# B&R Automation Studio project PickAndPlace
Automation Studio 6.3.1.32; Default project; technology packages: mappCockpit 6.3.1, mappMotion 6.4.1, mappView 6.3.1, mappVision 6.0.0, OpcUaCs 6.3.1

## Configuration APC3100

CPU 5APC3100.KBU3-000, AutomationRuntime 6.5.1, Build 11.3.0, Safety 0.0

### Task classes (Cpu.sw)
```
Cyclic#1 (cycle 2000 us, tolerance 0 us):
  Camera <- Tasks.Camera.prg
  BufferInit <- Tasks.BufferInit.prg
  Mechanics <- Tasks.Mechanics.prg
DataObjects: McAcpSys, assl1, Acp10sys, Arnc0sys
NcDataObjects: McDriveLog, gS_AxRepoi, gS_AxR1QCa, gS_AxR1QCi, gS_AxRepoa
Binaries: udbdef, arsvcreg, McMechSys, McAcpSim, McAcpDrv, TCData, mvLoader, McProfGen, mvConfig, OpcUaSrv, ViUnits, mCoWebSc, ashwac, Hierarchy, arconfig, ashwd, asfw, sysconf, iomap, Role, User, Settings, MechSys2, MechSys1, AxGrp1, Feat2, Axis2, Axis1, TrkPath, Feat1, AxGrp2, Ws2, Ws1, Conveyer, Config, Config_1, Config_2, TraceConfi, UaCsConfig, BRRole, Conveyor, TrkFrmSel1, TrkFrmSel2, viComp, Settings_1, viApp, viApp_1, FWRules, Config_3, ArFlatPrv, ArCoal, Config_8, vcpk, vcwxprt, vcpfar10, vcshared, vcfile, vcpfmtcx, arial, vcgclass, vcalarm, vcdsint, vcpfapc, arialbd, vcdsloc, vcmgr, vcbclass, StdVi102, StdVi101, StdVi103, StdVis02, StdVis03, StdVis01, vcnet, vctcal, vcpdihd, vcptusb, acp10cfg, Arnc0map, arnc0cfg, Acp10map, TCPmap, vcfntttf, vccbmp, SimVis01, vcrt, vcpdvnc, SimVis02, vcpdsw, vcpkat, vcctext, SimVis03, vccshape, vccbtn, vccovl, AdvVis03, AdvVis02, AdvVis01, vccstr, vccurl, vccbar, vcchtml, vccnum, vcxml, vccalarm, vcclbox, vccedit, Config_7, Config_6, Config_4, Config_5, TrkPath1
Libraries: Runtime, Operator, AsIecCon, astime, sys_lib, FileIO, AsMem, brsystem, AsBrStr, AsIOTime, standard, AsArSdm, AsBrWStr, AsZip, AsIO, AsHttp, AsIODiag, AsBrMath, MpBase, CoTrace, McBase, McAxGroup, McAcpAx, McAxis, McPathGen, McTrkPath, MpAxis, McProgInt, MpPick, McPureVAx, MpRobotics, MpTool, ViBase, AsARCfg, powerlnk, AsEPL, AsTCP, ArSsl, DataObj, UaCoal, AsArProf, UaCoalPrv, UaCore, ashw, vcresman
```

### Hardware
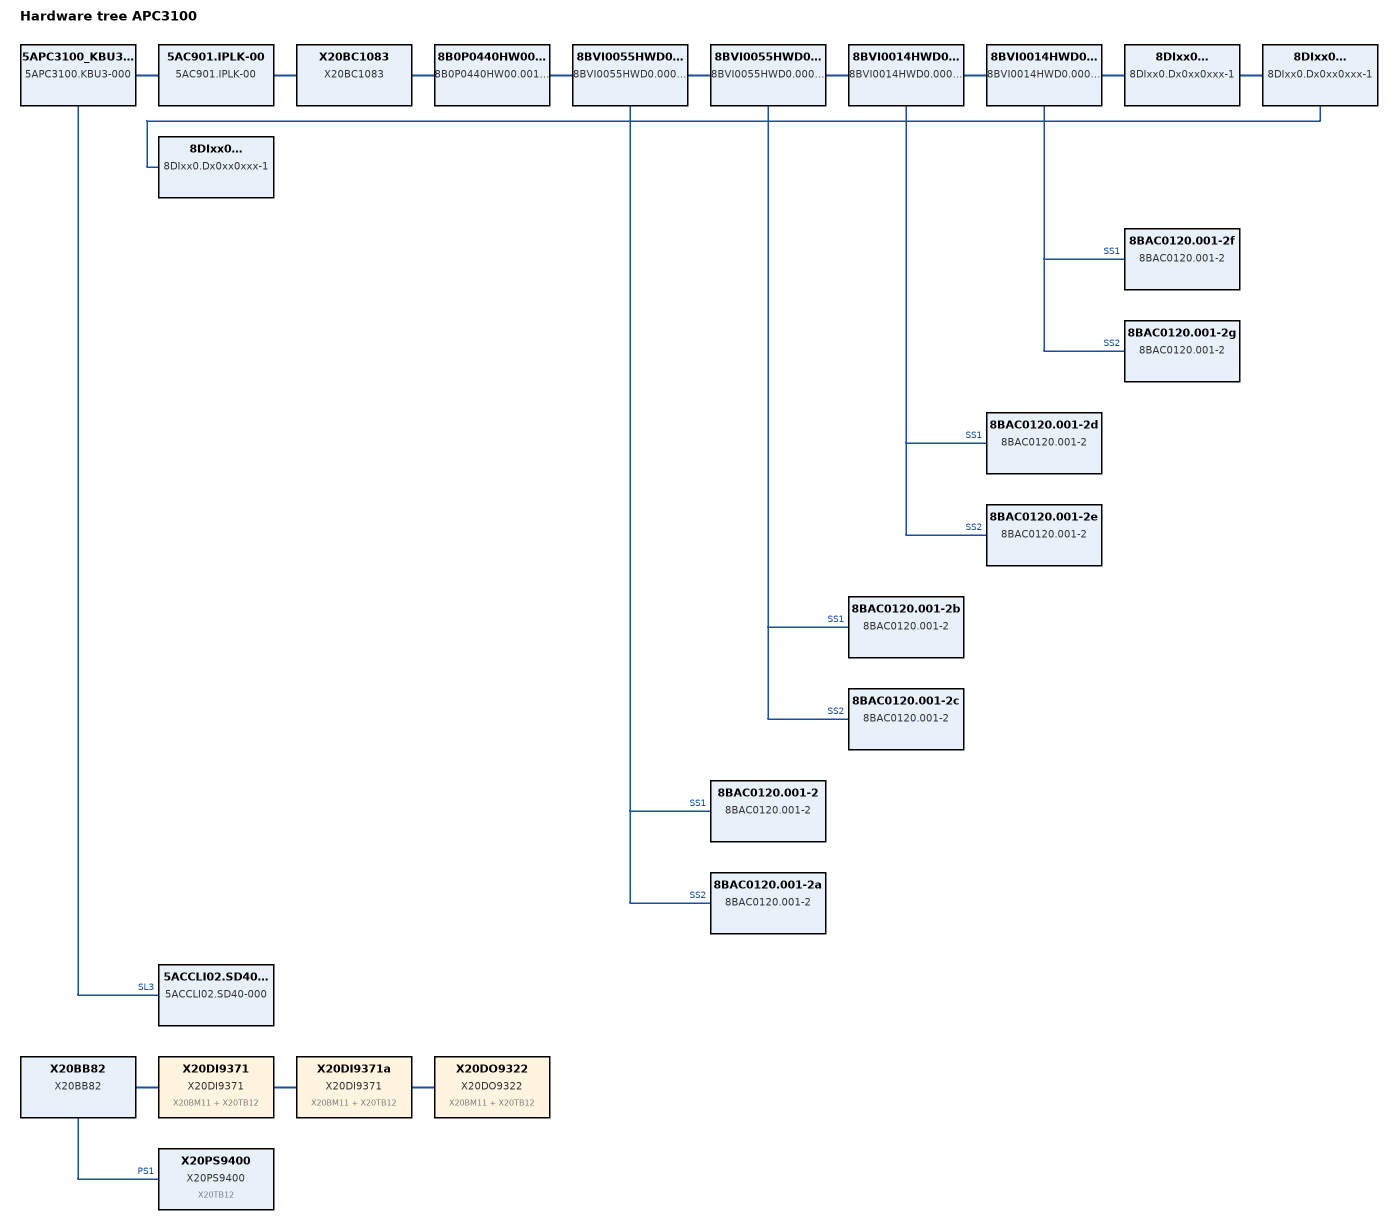
```
5AC901.IPLK-00 : 5AC901.IPLK-00 v2.1.0.0  [SL -> 5APC3100_KBU3_000.SL2]
  Connector IF1:
    MtuSize = 1500
    Channel1
    ChannelID1 = McAcpBroadcast
    ChannelType1 = OCTET[96]
    InternetAddress = 192.168.200.240
    SubnetMask = 255.255.255.0
    ActivateANSL = 1
    ActivateIpForwarding = 1
5ACCLI02.SD40-000 : 5ACCLI02.SD40-000 v2.1.0.0  [SL -> 5APC3100_KBU3_000.SL3]
  Supervision = off
5APC3100_KBU3_000 : 5APC3100.KBU3-000 v2.3.1.0
  Connector IF3:
    AssignedOperatingSystem = ARemb
    ActivateDevice = 1
    HostName = apc3100motorlabsbg
  Connector IF4:
    AssignedOperatingSystem = ARemb
    ActivateDevice = 1
    HostName = apc3100motorlabsbg
    Mode = Manual
    InternetAddress = 192.168.20.250
    SubnetMask = 255.255.255.0
    Vnc1
    VncTitle1 = VNC
    ActivateSnmp = 2
    ActivateIpForwarding = 1
  Connector IF5:
    AssignedOperatingSystem = ARemb
  Connector IF6:
    AssignedOperatingSystem = ARemb
  Connector IF7:
    AssignedOperatingSystem = ARemb
  Connector IF8:
    AssignedOperatingSystem = ARemb
  ConfigurationID = PickAndPlace_Real_APC910
  Simulation = 1
  RemMemDevice = PCI.2.IPLK.SRAM
  RemMemSize = 64000
  PermanentPvSize = 32000
  RemanentGlobalPvSize = 16000
  TimerDeviceType = EPLX2X
  TimerDevice = 5AC901.IPLK-00.IF1
  TaskClassIdleTime = 2000
  Cyclic1Duration = 2000
  Cyclic1Tolerance = 0
  Cyclic1Stack = 655360
  Cyclic1Output = 1
  Cyclic2Duration = 4000
  Cyclic2Tolerance = 4000
  Cyclic3Duration = 6000
  Cyclic3Tolerance = 6000
  Cyclic4Duration = 8000
  Cyclic4Tolerance = 8000
  Cyclic5Duration = 100000
  Cyclic5Tolerance = 100000
  FileDevice1
  FileDeviceName1 = RobotMotionPrgDir
  FileDevicePath1 = USER_PATH\..\..\..\..\..\Logical\UserPartitionData\RobotMotionPrgDir  // No simulation: use  USER_PATH\RobotMotionPrgDir   ;        Simulation: use    USER_PATH\..\..\..\..\..\Logical\UserPartitionData\RobotMotionPrgDir    to directly access the current progam state
  FileDevice2
  FileDeviceName2 = AutoGeneratedScene
  FileDevicePath2 = USER_PATH
  EthernetHostName = apc3100motorlabsbg
  ActivateFtpServer = 1
  FtpUser1
  FtpUsername1 = gmctest
  FtpUserPassword1 = qT0dlrKemp8H+/2V4GRHUzUq1qxdxChn7SWtcolMOPQ=
  FtpUserSalt1 = 1zGWL4Fu
  FTPAccessRight1 = 0
  ActivateWebServer = 1
  ActivateSdm = 1
8B0P0440HW00.001-1 : 8B0P0440HW00.001-1 v2.3.0.3 (NodeNumber=4)  [PLK1 -> X20BC1083.PLK2 [Cable Type=PowerlinkCable, Length=10, Version=1.0.0.3]; PLK2 -> 8BVI0055HWD0.000-1.PLK1 [Cable Type=PowerlinkCable, Length=10, Version=1.0.0.3]]
  DriveConfiguration/Module:
    McAcoposTypeID = AcoposMultiPSMpConfig
    ActivateACOPOSSimulationOnPLC = 0
    SWResetAfterFirmwareUpdate = 0
  DriveConfiguration/Channel[1]/PowerSection:
    AxisReference = gPsm
8BAC0120.001-2 : 8BAC0120.001-2 v2.2.0.0  [SS -> 8BVI0055HWD0.000-1.SS1]  // Delta 1 - Q1
  PlugInType = Encoder
  McAcoposTypeID = AcoposMultiPlugInConfig
8BAC0120.001-2a : 8BAC0120.001-2 v2.2.0.0  [SS -> 8BVI0055HWD0.000-1.SS2]  // Delta 1 - Q3
  PlugInType = Encoder
  McAcoposTypeID = AcoposMultiPlugInConfig
8BAC0120.001-2b : 8BAC0120.001-2 v2.2.0.0  [SS -> 8BVI0055HWD0.000-1a.SS1]  // Delta 1 - Q2
  PlugInType = Encoder
  McAcoposTypeID = AcoposMultiPlugInConfig
8BAC0120.001-2c : 8BAC0120.001-2 v2.2.0.0  [SS -> 8BVI0055HWD0.000-1a.SS2]  // Delta 1 - Qc
  PlugInType = Encoder
  McAcoposTypeID = AcoposMultiPlugInConfig
8BAC0120.001-2d : 8BAC0120.001-2 v2.2.0.0  [SS -> 8BVI0014HWD0.000-1.SS1]  // Delta 2 - Qc
  PlugInType = Encoder
  McAcoposTypeID = AcoposMultiPlugInConfig
8BAC0120.001-2e : 8BAC0120.001-2 v2.2.0.0  [SS -> 8BVI0014HWD0.000-1.SS2]  // Conveyer 1
  PlugInType = Encoder
  McAcoposTypeID = AcoposMultiPlugInConfig
8BAC0120.001-2f : 8BAC0120.001-2 v2.2.0.0  [SS -> 8BVI0014HWD0.000-1a.SS1]  // Conveyer 2
  PlugInType = Encoder
  McAcoposTypeID = AcoposMultiPlugInConfig
8BAC0120.001-2g : 8BAC0120.001-2 v2.2.0.0  [SS -> 8BVI0014HWD0.000-1a.SS2]  // Repository
  PlugInType = Encoder
  McAcoposTypeID = AcoposMultiPlugInConfig
8BVI0014HWD0.000-1 : 8BVI0014HWD0.000-1 v2.3.0.2 (NodeNumber=7)  [PLK1 -> 8BVI0055HWD0.000-1a.PLK2 [Cable Type=PowerlinkCable, Length=10, Version=1.0.0.3]; PLK2 -> 8BVI0014HWD0.000-1a.PLK1 [Cable Type=PowerlinkCable, Length=10, Version=1.0.0.3]]
  DriveConfiguration/Module:
    PowerSupply = DCBusVoltage
  DriveConfiguration/Module/PowerSupply:
    BusVoltage = 550
  DriveConfiguration/Channel[1]/RealAxis:
    AxisReference = delta2Qc
  DriveConfiguration/Channel[1]/RealAxis/MechanicalElements/Gearbox:
    Input = 10
  DriveConfiguration/Channel[1]/RealAxis/MechanicalElements/RotaryToLinearTransformation:
    ReferenceDistance = 3
  DriveConfiguration/Channel[1]/RealAxis/Controller/Mode/Position:
    ProportionalGain = 340
  DriveConfiguration/Channel[1]/RealAxis/Controller/Mode/Speed:
    ProportionalGain = 1.35
  DriveConfiguration/Channel[1]/RealAxis/Homing:
    Mode = Absolute
  DriveConfiguration/Channel[1]/RealAxis/Homing/Mode:
    Position = 14929.177
  DriveConfiguration/Channel[1]/RealAxis/Homing:
    RestorePositionVariable = 
  DriveConfiguration/Channel[1]/RealAxis/MovementErrorLimits:
    PositionError = 1.0
  DriveConfiguration/Channel[2]/RealAxis:
    AxisReference = conveyer1Ax
  DriveConfiguration/Channel[2]/RealAxis/MechanicalElements/Gearbox:
    Output = 10
  DriveConfiguration/Channel[2]/RealAxis/MechanicalElements/RotaryToLinearTransformation:
    ReferenceDistance = 3
  DriveConfiguration/Channel[2]/RealAxis/Controller/Mode/Position:
    ProportionalGain = 460
  DriveConfiguration/Channel[2]/RealAxis/Controller/Mode/Speed:
    ProportionalGain = 0.6
  DriveConfiguration/Channel[2]/RealAxis/Homing/Mode:
    Position = 5
  DriveConfiguration/Channel[2]/RealAxis/Homing:
    RestorePositionVariable = 
  DriveConfiguration/Channel[2]/RealAxis/MovementErrorLimits:
    PositionError = 1.0
  DriveConfiguration/Channel[2]/RealAxis/AxisFeatures:
    FeatureRef[1] = ProfGen
8BVI0014HWD0.000-1a : 8BVI0014HWD0.000-1 v2.3.0.2  [PLK1 -> 8BVI0014HWD0.000-1.PLK2 [Cable Type=PowerlinkCable, Length=10, Version=1.0.0.3]; PLK2 -> 8DIxx0.Dx0xx0xxx-1.PLK1 [Cable Type=PowerlinkCable, Length=10, Version=1.0.0.3]]
  DriveConfiguration/Module:
    PowerSupply = DCBusVoltage
  DriveConfiguration/Module/PowerSupply:
    BusVoltage = 550
  DriveConfiguration/Channel[1]/RealAxis:
    AxisReference = conveyer2Ax
  DriveConfiguration/Channel[1]/RealAxis/MechanicalElements/Gearbox:
    Output = 10
  DriveConfiguration/Channel[1]/RealAxis/MechanicalElements/RotaryToLinearTransformation:
    ReferenceDistance = 3
  DriveConfiguration/Channel[1]/RealAxis/Controller/Mode/Position:
    ProportionalGain = 420
  DriveConfiguration/Channel[1]/RealAxis/Controller/Mode/Speed:
    ProportionalGain = 0.55
  DriveConfiguration/Channel[1]/RealAxis/Homing/Mode:
    Position = 5
  DriveConfiguration/Channel[1]/RealAxis/Homing:
    RestorePositionVariable = 
  DriveConfiguration/Channel[1]/RealAxis/MovementErrorLimits:
    PositionError = 1.0
  DriveConfiguration/Channel[1]/RealAxis/AxisFeatures:
    FeatureRef[1] = ProfGen
  DriveConfiguration/Channel[2]/RealAxis:
    AxisReference = repositoryAx
  DriveConfiguration/Channel[2]/RealAxis/MechanicalElements/RotaryToLinearTransformation:
    ReferenceDistance = 16
  DriveConfiguration/Channel[2]/RealAxis/Controller/Mode/Position:
    ProportionalGain = 500.0
  DriveConfiguration/Channel[2]/RealAxis/Controller/Mode/Speed:
    ProportionalGain = 0.3
  DriveConfiguration/Channel[2]/RealAxis/Homing:
    Mode = Absolute
  DriveConfiguration/Channel[2]/RealAxis/Homing/Mode:
    Position = -58251.071
  DriveConfiguration/Channel[2]/RealAxis/Homing:
    RestorePositionVariable = 
  DriveConfiguration/Channel[2]/RealAxis/MovementErrorLimits:
    PositionError = 1.0
8BVI0055HWD0.000-1 : 8BVI0055HWD0.000-1 v2.3.0.2 (NodeNumber=5)  [PLK1 -> 8B0P0440HW00.001-1.PLK2 [Cable Type=PowerlinkCable, Length=10, Version=1.0.0.3]; PLK2 -> 8BVI0055HWD0.000-1a.PLK1 [Cable Type=PowerlinkCable, Length=10, Version=1.0.0.3]]
  DriveConfiguration/Module:
    McAcoposTypeID = AcoposMultiDConfig
    ActivateACOPOSSimulationOnPLC = 0
    PowerSupply = DCBusVoltage
  DriveConfiguration/Module/PowerSupply:
    BusVoltage = 550
  DriveConfiguration/Channel[1]/RealAxis:
    AxisReference = delta1Q1
    MechanicalElementsIsInvisible = 0
  DriveConfiguration/Channel[1]/RealAxis/MechanicalElements/Gearbox:
    InputIsReadOnly = 0
    Input = 31
    OutputIsReadOnly = 0
    Output = 1
  DriveConfiguration/Channel[1]/RealAxis/MechanicalElements/RotaryToLinearTransformation:
    ReferenceDistanceIsReadOnly = 0
    ReferenceDistance = 1
  DriveConfiguration/Channel[1]/RealAxis/Controller:
    ModeIsReadOnly = 0
    Mode = PositionController
  DriveConfiguration/Channel[1]/RealAxis/Controller/Mode/Position:
    ProportionalGain = 420
    IntegrationTime = 0.0
    PredictionTime = 0.0004
    TotalDelayTime = 0.0004
  DriveConfiguration/Channel[1]/RealAxis/Controller/Mode/Speed:
    ProportionalGainIsReadOnly = 0
    ProportionalGain = 1.65
    IntegrationTimeIsReadOnly = 0
    IntegrationTime = 0.0
    FilterTimeIsReadOnly = 0
    FilterTime = 0.0
  DriveConfiguration/Channel[1]/RealAxis/Controller/Mode/LoopFilters:
    LoopFilterXIsReadOnly = 0
    LoopFilter1 = NotUsed
    LoopFilter2 = NotUsed
    LoopFilter3 = NotUsed
  DriveConfiguration/Channel[1]/RealAxis/Homing:
    ModeIsReadOnly = 0
    Mode = Absolute
  DriveConfiguration/Channel[1]/RealAxis/Homing/Mode:
    Position = 17776.525
  DriveConfiguration/Channel[1]/RealAxis/Homing:
    RestorePositionVariable = 
  DriveConfiguration/Channel[1]/RealAxis/StopReaction:
    QuickstopIsReadOnly = 0
    Quickstop = DecelerationLimit
    DriveErrorIsReadOnly = 0
    DriveError = DecelerationLimit
  DriveConfiguration/Channel[1]/RealAxis/MovementErrorLimits:
    PositionError = 1.0
    VelocityErrorMonitoring = Automatic1
  DriveConfiguration/Channel[1]/RealAxis:
    JerkFilterIsReadOnly = 0
    JerkFilter = NotUsed
    ZeroVibrationFilter = NotUsed
  DriveConfiguration/Channel[1]/RealAxis/DigitalInputs/HomingSwitch:
    SourceIsReadOnly = 0
    Source = NotUsed
    Level = High
  DriveConfiguration/Channel[1]/RealAxis/DigitalInputs/PositiveLimitSwitch:
    SourceIsReadOnly = 0
    Source = NotUsed
    Level = High
  DriveConfiguration/Channel[1]/RealAxis/DigitalInputs/NegativeLimitSwitch:
    SourceIsReadOnly = 0
    Source = NotUsed
    Level = High
  DriveConfiguration/Channel[1]/RealAxis/DigitalInputs/Trigger1:
    Source = X2Trigger1
    Level = High
  DriveConfiguration/Channel[1]/RealAxis/DigitalInputs/Trigger2:
    Source = X2Trigger2
    Level = High
  DriveConfiguration/Channel[1]/RealAxis/DigitalInputs/Quickstop:
    Input = Trigger2
  DriveConfiguration/Channel[1]/RealAxis/Simulation:
    SimulationModeOnPLC = SetValueGeneration
    SimulationModeOnACOPOS = NotUsed
  DriveConfiguration/Channel[1]:
    ExternalEncoderAxis = NotUsed
  DriveConfiguration/Channel[2]/RealAxis:
    AxisReference = delta1Q3
    MechanicalElementsIsInvisible = 0
  DriveConfiguration/Channel[2]/RealAxis/MechanicalElements/Gearbox:
    InputIsReadOnly = 0
    Input = 31
    OutputIsReadOnly = 0
    Output = 1
  DriveConfiguration/Channel[2]/RealAxis/MechanicalElements/RotaryToLinearTransformation:
    ReferenceDistanceIsReadOnly = 0
    ReferenceDistance = 1
  DriveConfiguration/Channel[2]/RealAxis/Controller:
    ModeIsReadOnly = 0
    Mode = PositionController
  DriveConfiguration/Channel[2]/RealAxis/Controller/Mode/Position:
    ProportionalGain = 420
    IntegrationTime = 0.0
    PredictionTime = 0.0004
    TotalDelayTime = 0.0004
  DriveConfiguration/Channel[2]/RealAxis/Controller/Mode/Speed:
    ProportionalGainIsReadOnly = 0
    ProportionalGain = 1.65
    IntegrationTimeIsReadOnly = 0
    IntegrationTime = 0.0
    FilterTimeIsReadOnly = 0
    FilterTime = 0.0
  DriveConfiguration/Channel[2]/RealAxis/Controller/Mode/LoopFilters:
    LoopFilterXIsReadOnly = 0
    LoopFilter1 = NotUsed
    LoopFilter2 = NotUsed
    LoopFilter3 = NotUsed
  DriveConfiguration/Channel[2]/RealAxis/Homing:
    ModeIsReadOnly = 0
    Mode = Absolute
  DriveConfiguration/Channel[2]/RealAxis/Homing/Mode:
    Position = 44644.06
  DriveConfiguration/Channel[2]/RealAxis/Homing:
    RestorePositionVariable = 
  DriveConfiguration/Channel[2]/RealAxis/StopReaction:
    QuickstopIsReadOnly = 0
    Quickstop = DecelerationLimit
    DriveErrorIsReadOnly = 0
    DriveError = DecelerationLimit
  DriveConfiguration/Channel[2]/RealAxis/MovementErrorLimits:
    PositionError = 1.0
    VelocityErrorMonitoring = Automatic1
  DriveConfiguration/Channel[2]/RealAxis:
    JerkFilterIsReadOnly = 0
    JerkFilter = NotUsed
    ZeroVibrationFilter = NotUsed
  DriveConfiguration/Channel[2]/RealAxis/DigitalInputs/HomingSwitch:
    SourceIsReadOnly = 0
    Source = NotUsed
    Level = High
  DriveConfiguration/Channel[2]/RealAxis/DigitalInputs/PositiveLimitSwitch:
    SourceIsReadOnly = 0
    Source = NotUsed
    Level = High
  DriveConfiguration/Channel[2]/RealAxis/DigitalInputs/NegativeLimitSwitch:
    SourceIsReadOnly = 0
    Source = NotUsed
    Level = High
  DriveConfiguration/Channel[2]/RealAxis/DigitalInputs/Trigger1:
    Source = X2Trigger1
    Level = High
  DriveConfiguration/Channel[2]/RealAxis/DigitalInputs/Trigger2:
    Source = X2Trigger2
    Level = High
  DriveConfiguration/Channel[2]/RealAxis/DigitalInputs/Quickstop:
    Input = Trigger2
  DriveConfiguration/Channel[2]/RealAxis/Simulation:
    SimulationModeOnPLC = SetValueGeneration
    SimulationModeOnACOPOS = NotUsed
  DriveConfiguration/Channel[2]:
    ExternalEncoderAxis = NotUsed
8BVI0055HWD0.000-1a : 8BVI0055HWD0.000-1 v2.3.0.2 (NodeNumber=6)  [PLK1 -> 8BVI0055HWD0.000-1.PLK2 [Cable Type=PowerlinkCable, Length=10, Version=1.0.0.3]; PLK2 -> 8BVI0014HWD0.000-1.PLK1 [Cable Type=PowerlinkCable, Length=10, Version=1.0.0.3]]
  DriveConfiguration/Module:
    McAcoposTypeID = AcoposMultiDConfig
    ActivateACOPOSSimulationOnPLC = 0
    PowerSupply = DCBusVoltage
  DriveConfiguration/Module/PowerSupply:
    BusVoltage = 550
  DriveConfiguration/Channel[1]/RealAxis:
    AxisReference = delta1Q2
    MechanicalElementsIsInvisible = 0
  DriveConfiguration/Channel[1]/RealAxis/MechanicalElements/Gearbox:
    InputIsReadOnly = 0
    Input = 31
    OutputIsReadOnly = 0
    Output = 1
  DriveConfiguration/Channel[1]/RealAxis/MechanicalElements/RotaryToLinearTransformation:
    ReferenceDistanceIsReadOnly = 0
    ReferenceDistance = 1
  DriveConfiguration/Channel[1]/RealAxis/Controller:
    ModeIsReadOnly = 0
    Mode = PositionController
  DriveConfiguration/Channel[1]/RealAxis/Controller/Mode/Position:
    ProportionalGain = 420
    IntegrationTime = 0.0
    PredictionTime = 0.0004
    TotalDelayTime = 0.0004
  DriveConfiguration/Channel[1]/RealAxis/Controller/Mode/Speed:
    ProportionalGainIsReadOnly = 0
    ProportionalGain = 1.65
    IntegrationTimeIsReadOnly = 0
    IntegrationTime = 0.0
    FilterTimeIsReadOnly = 0
    FilterTime = 0.0
  DriveConfiguration/Channel[1]/RealAxis/Controller/Mode/LoopFilters:
    LoopFilterXIsReadOnly = 0
    LoopFilter1 = NotUsed
    LoopFilter2 = NotUsed
    LoopFilter3 = NotUsed
  DriveConfiguration/Channel[1]/RealAxis/Homing:
    ModeIsReadOnly = 0
    Mode = Absolute
  DriveConfiguration/Channel[1]/RealAxis/Homing/Mode:
    Position = 26128.766
  DriveConfiguration/Channel[1]/RealAxis/Homing:
    RestorePositionVariable = 
  DriveConfiguration/Channel[1]/RealAxis/StopReaction:
    QuickstopIsReadOnly = 0
    Quickstop = DecelerationLimit
    DriveErrorIsReadOnly = 0
    DriveError = DecelerationLimit
  DriveConfiguration/Channel[1]/RealAxis/MovementErrorLimits:
    PositionError = 1.0
    VelocityErrorMonitoring = Automatic1
  DriveConfiguration/Channel[1]/RealAxis:
    JerkFilterIsReadOnly = 0
    JerkFilter = NotUsed
    ZeroVibrationFilter = NotUsed
  DriveConfiguration/Channel[1]/RealAxis/DigitalInputs/HomingSwitch:
    SourceIsReadOnly = 0
    Source = NotUsed
    Level = High
  DriveConfiguration/Channel[1]/RealAxis/DigitalInputs/PositiveLimitSwitch:
    SourceIsReadOnly = 0
    Source = NotUsed
    Level = High
  DriveConfiguration/Channel[1]/RealAxis/DigitalInputs/NegativeLimitSwitch:
    SourceIsReadOnly = 0
    Source = NotUsed
    Level = High
  DriveConfiguration/Channel[1]/RealAxis/DigitalInputs/Trigger1:
    Source = X2Trigger1
    Level = High
  DriveConfiguration/Channel[1]/RealAxis/DigitalInputs/Trigger2:
    Source = X2Trigger2
    Level = High
  DriveConfiguration/Channel[1]/RealAxis/DigitalInputs/Quickstop:
    Input = Trigger2
  DriveConfiguration/Channel[1]/RealAxis/Simulation:
    SimulationModeOnPLC = SetValueGeneration
    SimulationModeOnACOPOS = NotUsed
  DriveConfiguration/Channel[1]:
    ExternalEncoderAxis = NotUsed
  DriveConfiguration/Channel[2]/RealAxis:
    AxisReference = delta1Qc
    MechanicalElementsIsInvisible = 0
  DriveConfiguration/Channel[2]/RealAxis/MechanicalElements/Gearbox:
    InputIsReadOnly = 0
    Input = 10
    OutputIsReadOnly = 0
    Output = 1
  DriveConfiguration/Channel[2]/RealAxis/MechanicalElements/RotaryToLinearTransformation:
    ReferenceDistanceIsReadOnly = 0
    ReferenceDistance = 1
  DriveConfiguration/Channel[2]/RealAxis/Controller:
    ModeIsReadOnly = 0
    Mode = PositionController
  DriveConfiguration/Channel[2]/RealAxis/Controller/Mode/Position:
    ProportionalGain = 400
    IntegrationTime = 0.0
    PredictionTime = 0.0004
    TotalDelayTime = 0.0004
  DriveConfiguration/Channel[2]/RealAxis/Controller/Mode/Speed:
    ProportionalGainIsReadOnly = 0
    ProportionalGain = 1.2
    IntegrationTimeIsReadOnly = 0
    IntegrationTime = 0.0
    FilterTimeIsReadOnly = 0
    FilterTime = 0.0
  DriveConfiguration/Channel[2]/RealAxis/Controller/Mode/LoopFilters:
    LoopFilterXIsReadOnly = 0
    LoopFilter1 = NotUsed
    LoopFilter2 = NotUsed
    LoopFilter3 = NotUsed
  DriveConfiguration/Channel[2]/RealAxis/Homing:
    ModeIsReadOnly = 0
    Mode = Absolute
  DriveConfiguration/Channel[2]/RealAxis/Homing/Mode:
    Position = 68668.338
  DriveConfiguration/Channel[2]/RealAxis/Homing:
    RestorePositionVariable = 
  DriveConfiguration/Channel[2]/RealAxis/StopReaction:
    QuickstopIsReadOnly = 0
    Quickstop = DecelerationLimit
    DriveErrorIsReadOnly = 0
    DriveError = DecelerationLimit
  DriveConfiguration/Channel[2]/RealAxis/MovementErrorLimits:
    PositionError = 1.0
    VelocityErrorMonitoring = Automatic1
  DriveConfiguration/Channel[2]/RealAxis:
    JerkFilterIsReadOnly = 0
    JerkFilter = NotUsed
    ZeroVibrationFilter = NotUsed
  DriveConfiguration/Channel[2]/RealAxis/DigitalInputs/HomingSwitch:
    SourceIsReadOnly = 0
    Source = NotUsed
    Level = High
  DriveConfiguration/Channel[2]/RealAxis/DigitalInputs/PositiveLimitSwitch:
    SourceIsReadOnly = 0
    Source = NotUsed
    Level = High
  DriveConfiguration/Channel[2]/RealAxis/DigitalInputs/NegativeLimitSwitch:
    SourceIsReadOnly = 0
    Source = NotUsed
    Level = High
  DriveConfiguration/Channel[2]/RealAxis/DigitalInputs/Trigger1:
    Source = X2Trigger1
    Level = High
  DriveConfiguration/Channel[2]/RealAxis/DigitalInputs/Trigger2:
    Source = X2Trigger2
    Level = High
  DriveConfiguration/Channel[2]/RealAxis/DigitalInputs/Quickstop:
    Input = Trigger2
  DriveConfiguration/Channel[2]/RealAxis/Simulation:
    SimulationModeOnPLC = SetValueGeneration
    SimulationModeOnACOPOS = NotUsed
  DriveConfiguration/Channel[2]:
    ExternalEncoderAxis = NotUsed
8DIxx0.Dx0xx0xxx-1 : 8DIxx0.Dx0xx0xxx-1 v2.3.0.2 (NodeNumber=9)  [PLK1 -> 8BVI0014HWD0.000-1a.PLK2 [Cable Type=PowerlinkCable, Length=10, Version=1.0.0.3]; PLK2 -> 8DIxx0.Dx0xx0xxx-1a.PLK1 [Cable Type=PowerlinkCable, Length=10, Version=1.0.0.3]]  // Delta 2 - Q1
  DriveConfiguration/Module:
    McAcoposTypeID = AcoposMotorConfig
    ActivateACOPOSSimulationOnPLC = 0
  DriveConfiguration/Module/PowerSupply:
    PowerSupplyModuleReference = gPsm
  DriveConfiguration/Channel[1]/RealAxis:
    AxisReference = delta2Q1
    MechanicalElementsIsInvisible = 0
  DriveConfiguration/Channel[1]/RealAxis/MechanicalElements/Gearbox:
    InputIsReadOnly = 0
    Input = 31
    OutputIsReadOnly = 0
    Output = 1
  DriveConfiguration/Channel[1]/RealAxis/MechanicalElements/RotaryToLinearTransformation:
    ReferenceDistanceIsReadOnly = 0
    ReferenceDistance = 1
  DriveConfiguration/Channel[1]/RealAxis/Controller:
    ModeIsReadOnly = 0
    Mode = PositionController
  DriveConfiguration/Channel[1]/RealAxis/Controller/Mode/Position:
    ProportionalGain = 460
    IntegrationTime = 0.0
    PredictionTime = 0.0004
    TotalDelayTime = 0.0004
  DriveConfiguration/Channel[1]/RealAxis/Controller/Mode/Speed:
    ProportionalGainIsReadOnly = 0
    ProportionalGain = 1.2
    IntegrationTimeIsReadOnly = 0
    IntegrationTime = 0.0
    FilterTimeIsReadOnly = 0
    FilterTime = 0.0
  DriveConfiguration/Channel[1]/RealAxis/Controller/Mode/LoopFilters:
    LoopFilterXIsReadOnly = 0
    LoopFilter1 = NotUsed
    LoopFilter2 = NotUsed
    LoopFilter3 = NotUsed
  DriveConfiguration/Channel[1]/RealAxis/Homing:
    ModeIsReadOnly = 0
    Mode = Absolute
  DriveConfiguration/Channel[1]/RealAxis/Homing/Mode:
    Position = 39202.357
  DriveConfiguration/Channel[1]/RealAxis/Homing:
    RestorePositionVariable = 
  DriveConfiguration/Channel[1]/RealAxis/StopReaction:
    QuickstopIsReadOnly = 0
    Quickstop = DecelerationLimit
    DriveErrorIsReadOnly = 0
    DriveError = DecelerationLimit
  DriveConfiguration/Channel[1]/RealAxis/MovementErrorLimits:
    PositionError = 1.0
    VelocityErrorMonitoring = Automatic1
  DriveConfiguration/Channel[1]/RealAxis:
    JerkFilterIsReadOnly = 0
    JerkFilter = NotUsed
    ZeroVibrationFilter = NotUsed
  DriveConfiguration/Channel[1]/RealAxis/DigitalInputs/HomingSwitch:
    SourceIsReadOnly = 0
    Source = X1Ref
    Level = High
  DriveConfiguration/Channel[1]/RealAxis/DigitalInputs/PositiveLimitSwitch:
    Source = X1PosLim
    Level = High
  DriveConfiguration/Channel[1]/RealAxis/DigitalInputs/NegativeLimitSwitch:
    Source = X1NegLim
    Level = High
  DriveConfiguration/Channel[1]/RealAxis/DigitalInputs/Trigger1:
    Source = X1Trigger1
    Level = High
  DriveConfiguration/Channel[1]/RealAxis/DigitalInputs/Trigger2:
    Source = X1Trigger2
    Level = High
  DriveConfiguration/Channel[1]/RealAxis/DigitalInputs/Quickstop:
    Input = Trigger2
  DriveConfiguration/Channel[1]/RealAxis/Simulation:
    SimulationModeOnPLC = SetValueGeneration
    SimulationModeOnACOPOS = NotUsed
8DIxx0.Dx0xx0xxx-1a : 8DIxx0.Dx0xx0xxx-1 v2.3.0.2 (NodeNumber=10)  [PLK1 -> 8DIxx0.Dx0xx0xxx-1.PLK2 [Cable Type=PowerlinkCable, Length=10, Version=1.0.0.3]; PLK2 -> 8DIxx0.Dx0xx0xxx-1b.PLK1 [Cable Type=PowerlinkCable, Length=10, Version=1.0.0.3]]  // Delta 2 - Q2
  DriveConfiguration/Module:
    McAcoposTypeID = AcoposMotorConfig
    ActivateACOPOSSimulationOnPLC = 0
  DriveConfiguration/Module/PowerSupply:
    PowerSupplyModuleReference = gPsm
  DriveConfiguration/Channel[1]/RealAxis:
    AxisReference = delta2Q2
    MechanicalElementsIsInvisible = 0
  DriveConfiguration/Channel[1]/RealAxis/MechanicalElements/Gearbox:
    InputIsReadOnly = 0
    Input = 31
    OutputIsReadOnly = 0
    Output = 1
  DriveConfiguration/Channel[1]/RealAxis/MechanicalElements/RotaryToLinearTransformation:
    ReferenceDistanceIsReadOnly = 0
    ReferenceDistance = 1
  DriveConfiguration/Channel[1]/RealAxis/Controller:
    ModeIsReadOnly = 0
    Mode = PositionController
  DriveConfiguration/Channel[1]/RealAxis/Controller/Mode/Position:
    ProportionalGain = 600
    IntegrationTime = 0.0
    PredictionTime = 0.0004
    TotalDelayTime = 0.0004
  DriveConfiguration/Channel[1]/RealAxis/Controller/Mode/Speed:
    ProportionalGainIsReadOnly = 0
    ProportionalGain = 1.5
    IntegrationTimeIsReadOnly = 0
    IntegrationTime = 0.0
    FilterTimeIsReadOnly = 0
    FilterTime = 0.0
  DriveConfiguration/Channel[1]/RealAxis/Controller/Mode/LoopFilters:
    LoopFilterXIsReadOnly = 0
    LoopFilter1 = NotUsed
    LoopFilter2 = NotUsed
    LoopFilter3 = NotUsed
  DriveConfiguration/Channel[1]/RealAxis/Homing:
    ModeIsReadOnly = 0
    Mode = Absolute
  DriveConfiguration/Channel[1]/RealAxis/Homing/Mode:
    Position = 27322.805
  DriveConfiguration/Channel[1]/RealAxis/Homing:
    RestorePositionVariable = 
  DriveConfiguration/Channel[1]/RealAxis/StopReaction:
    QuickstopIsReadOnly = 0
    Quickstop = DecelerationLimit
    DriveErrorIsReadOnly = 0
    DriveError = DecelerationLimit
  DriveConfiguration/Channel[1]/RealAxis/MovementErrorLimits:
    PositionError = 1.0
    VelocityErrorMonitoring = Automatic1
  DriveConfiguration/Channel[1]/RealAxis:
    JerkFilterIsReadOnly = 0
    JerkFilter = NotUsed
    ZeroVibrationFilter = NotUsed
  DriveConfiguration/Channel[1]/RealAxis/DigitalInputs/HomingSwitch:
    SourceIsReadOnly = 0
    Source = X1Ref
    Level = High
  DriveConfiguration/Channel[1]/RealAxis/DigitalInputs/PositiveLimitSwitch:
    Source = X1PosLim
    Level = High
  DriveConfiguration/Channel[1]/RealAxis/DigitalInputs/NegativeLimitSwitch:
    Source = X1NegLim
    Level = High
  DriveConfiguration/Channel[1]/RealAxis/DigitalInputs/Trigger1:
    Source = X1Trigger1
    Level = High
  DriveConfiguration/Channel[1]/RealAxis/DigitalInputs/Trigger2:
    Source = X1Trigger2
    Level = High
  DriveConfiguration/Channel[1]/RealAxis/DigitalInputs/Quickstop:
    Input = Trigger2
  DriveConfiguration/Channel[1]/RealAxis/Simulation:
    SimulationModeOnPLC = SetValueGeneration
    SimulationModeOnACOPOS = NotUsed
8DIxx0.Dx0xx0xxx-1b : 8DIxx0.Dx0xx0xxx-1 v2.3.0.2 (NodeNumber=11)  [PLK1 -> 8DIxx0.Dx0xx0xxx-1a.PLK2 [Cable Type=PowerlinkCable, Length=10, Version=1.0.0.3]]  // Delta 2 - Q3
  DriveConfiguration/Module:
    McAcoposTypeID = AcoposMotorConfig
    ActivateACOPOSSimulationOnPLC = 0
  DriveConfiguration/Module/PowerSupply:
    PowerSupplyModuleReference = gPsm
  DriveConfiguration/Channel[1]/RealAxis:
    AxisReference = delta2Q3
    MechanicalElementsIsInvisible = 0
  DriveConfiguration/Channel[1]/RealAxis/MechanicalElements/Gearbox:
    InputIsReadOnly = 0
    Input = 31
    OutputIsReadOnly = 0
    Output = 1
  DriveConfiguration/Channel[1]/RealAxis/MechanicalElements/RotaryToLinearTransformation:
    ReferenceDistanceIsReadOnly = 0
    ReferenceDistance = 1
  DriveConfiguration/Channel[1]/RealAxis/Controller:
    ModeIsReadOnly = 0
    Mode = PositionController
  DriveConfiguration/Channel[1]/RealAxis/Controller/Mode/Position:
    ProportionalGain = 580
    IntegrationTime = 0.0
    PredictionTime = 0.0004
    TotalDelayTime = 0.0004
  DriveConfiguration/Channel[1]/RealAxis/Controller/Mode/Speed:
    ProportionalGainIsReadOnly = 0
    ProportionalGain = 1.45
    IntegrationTimeIsReadOnly = 0
    IntegrationTime = 0.0
    FilterTimeIsReadOnly = 0
    FilterTime = 0.0
  DriveConfiguration/Channel[1]/RealAxis/Controller/Mode/LoopFilters:
    LoopFilterXIsReadOnly = 0
    LoopFilter1 = NotUsed
    LoopFilter2 = NotUsed
    LoopFilter3 = NotUsed
  DriveConfiguration/Channel[1]/RealAxis/Homing:
    ModeIsReadOnly = 0
    Mode = Absolute
  DriveConfiguration/Channel[1]/RealAxis/Homing/Mode:
    Position = 35631.62
  DriveConfiguration/Channel[1]/RealAxis/Homing:
    RestorePositionVariable = 
  DriveConfiguration/Channel[1]/RealAxis/StopReaction:
    QuickstopIsReadOnly = 0
    Quickstop = DecelerationLimit
    DriveErrorIsReadOnly = 0
    DriveError = DecelerationLimit
  DriveConfiguration/Channel[1]/RealAxis/MovementErrorLimits:
    PositionError = 1.0
    VelocityErrorMonitoring = Automatic1
  DriveConfiguration/Channel[1]/RealAxis:
    JerkFilterIsReadOnly = 0
    JerkFilter = NotUsed
    ZeroVibrationFilter = NotUsed
  DriveConfiguration/Channel[1]/RealAxis/DigitalInputs/HomingSwitch:
    SourceIsReadOnly = 0
    Source = X1Ref
    Level = High
  DriveConfiguration/Channel[1]/RealAxis/DigitalInputs/PositiveLimitSwitch:
    Source = X1PosLim
    Level = High
  DriveConfiguration/Channel[1]/RealAxis/DigitalInputs/NegativeLimitSwitch:
    Source = X1NegLim
    Level = High
  DriveConfiguration/Channel[1]/RealAxis/DigitalInputs/Trigger1:
    Source = X1Trigger1
    Level = High
  DriveConfiguration/Channel[1]/RealAxis/DigitalInputs/Trigger2:
    Source = X1Trigger2
    Level = High
  DriveConfiguration/Channel[1]/RealAxis/DigitalInputs/Quickstop:
    Input = Trigger2
  DriveConfiguration/Channel[1]/RealAxis/Simulation:
    SimulationModeOnPLC = SetValueGeneration
    SimulationModeOnACOPOS = NotUsed
X20BB82 : X20BB82 v1.2.0.0
  Connector IF1:
    CycleTime = 1600
X20BC1083 : X20BC1083 v2.17.0.0 (NodeNumber=2)  [PLK1 -> 5AC901.IPLK-00.IF1 [Cable Type=PowerlinkCable, Length=10, Version=1.0.0.3]; PLK2 -> 8B0P0440HW00.001-1.PLK1 [Cable Type=PowerlinkCable, Length=10, Version=1.0.0.3]; SL -> X20BB82.SL1]
  Supervision = off
X20BM11 : X20BM11 v1.1.0.0  [X2X1 -> X20BB82.IF1]
X20BM11a : X20BM11 v1.1.0.0  [X2X1 -> X20BM11.X2X2]
X20BM11b : X20BM11 v1.1.0.0  [X2X1 -> X20BM11a.X2X2]
X20DI9371 : X20DI9371 v1.6.1.0  [SS1 -> X20TB12a.SS; SL -> X20BM11.SL1]
  Supervision = off
X20DI9371a : X20DI9371 v1.6.1.0  [SS1 -> X20TB12f.SS; SL -> X20BM11a.SL1]
  Supervision = off
X20DO9322 : X20DO9322 v1.7.0.0  [SS1 -> X20TB12c.SS; SL -> X20BM11b.SL1]
  Supervision = off
X20PS9400 : X20PS9400 v1.9.0.0  [SS1 -> X20TB12.SS; PS -> X20BB82.PS1]
  Supervision = off
X20TB12 : X20TB12 v1.0.0.0
X20TB12a : X20TB12 v1.0.0.0
X20TB12c : X20TB12 v1.0.0.0
X20TB12f : X20TB12 v1.0.0.0
```

### IoMap.iom - 5APC3100_KBU3_000/IoMap.iom
```iecst
(********************************************************************
 * COPYRIGHT -- Bernecker + Rainer
 ********************************************************************
 * File: IoMap.iom
 * Author: rognerp
 * Created: September 24, 2014
 ********************************************************************
 * IO mapping file
 ********************************************************************)
VAR_CONFIG
	::Mechanics:MotionProgramRob1.CloseGripper AT %QX."X20DO9322".DigitalOutput01;
	::Mechanics:MotionProgramRob2.CloseGripper AT %QX."X20DO9322".DigitalOutput02;
	::Mechanics:MotionProgramRob2.CloseGripper AT %QX."X20DO9322".DigitalOutput03;
	::Mechanics:MotionProgramRob2.CloseGripper AT %QX."X20DO9322".DigitalOutput04;
	::Mechanics:MotionProgramRob2.CloseGripper AT %QX."X20DO9322".DigitalOutput05;
	::Camera:CameraPV.Param.GainLevel AT %QB."VSC122R21.051P-000".GainLevel;
	::Camera:CameraPV.Param.SetFocus AT %QW."VSC122R21.051P-000".SetFocus;
	::Camera:CameraPV.Param.ExposureTime AT %QD."VSC122R21.051P-000".ExposureTime01;
	::Camera:CameraPV.Param.FlashColor AT %QB."VSC122R21.051P-000".FlashColor01;
	::Camera:CameraPV.Param.FlashSegment AT %QB."VSC122R21.051P-000".FlashSegment01;
	::Camera:CameraPV.Status.ModuleOk AT %IX."VSC122R21.051P-000".ModuleOk;
	::Camera:CameraPV.Status.CameraStatus AT %ID."VSC122R21.051P-000".CameraStatus;
	::Camera:CameraPV.Input.EnableVF AT %QX."VSC122R21.051P-000".Enable;
	::Camera:CameraPV.Input.NumSearchMax AT %QB."VSC122R21.051P-000".NumSearchMax;
	::Camera:CameraPV.Output.NumObjFound AT %IB."VSC122R21.051P-000".NumObjFound;
	::Camera:CameraPV.Output.Obj[0].Model AT %IB."VSC122R21.051P-000".Model01;
	::Camera:CameraPV.Output.Obj[1].Model AT %IB."VSC122R21.051P-000".Model02;
	::Camera:CameraPV.Output.Obj[2].Model AT %IB."VSC122R21.051P-000".Model03;
	::Camera:CameraPV.Output.Obj[3].Model AT %IB."VSC122R21.051P-000".Model04;
	::Camera:CameraPV.Output.Obj[0].Pos.X AT %ID."VSC122R21.051P-000".Pos_x01;
	::Camera:CameraPV.Output.Obj[0].Pos.Y AT %ID."VSC122R21.051P-000".Pos_y01;
	::Camera:CameraPV.Output.Obj[1].Pos.X AT %ID."VSC122R21.051P-000".Pos_x02;
	::Camera:CameraPV.Output.Obj[2].Pos.X AT %ID."VSC122R21.051P-000".Pos_x03;
	::Camera:CameraPV.Output.Obj[3].Pos.X AT %ID."VSC122R21.051P-000".Pos_x04;
	::Camera:CameraPV.Output.Obj[1].Pos.Y AT %ID."VSC122R21.051P-000".Pos_y02;
	::Camera:CameraPV.Output.Obj[2].Pos.Y AT %ID."VSC122R21.051P-000".Pos_y03;
	::Camera:CameraPV.Output.Obj[3].Pos.Y AT %ID."VSC122R21.051P-000".Pos_y04;
	::Camera:CameraPV.Status.CompletedAcquisitionCount AT %IB."VSC122R21.051P-000".CompletedAcquisitionCnt;
	::Camera:CameraPV.Status.ImageProcessingActive AT %IX."VSC122R21.051P-000".ImageProcessingActive;
	::Camera:CameraPV.Output.Obj[4].Model AT %IB."VSC122R21.051P-000".Model05;
	::Camera:CameraPV.Output.Obj[5].Model AT %IB."VSC122R21.051P-000".Model06;
	::Camera:CameraPV.Output.Obj[6].Model AT %IB."VSC122R21.051P-000".Model07;
	::Camera:CameraPV.Output.Obj[4].Pos.X AT %ID."VSC122R21.051P-000".Pos_x05;
	::Camera:CameraPV.Output.Obj[5].Pos.X AT %ID."VSC122R21.051P-000".Pos_x06;
	::Camera:CameraPV.Output.Obj[6].Pos.X AT %ID."VSC122R21.051P-000".Pos_x07;
	::Camera:CameraPV.Output.Obj[4].Pos.Y AT %ID."VSC122R21.051P-000".Pos_y05;
	::Camera:CameraPV.Output.Obj[5].Pos.Y AT %ID."VSC122R21.051P-000".Pos_y06;
	::Camera:CameraPV.Output.Obj[6].Pos.Y AT %ID."VSC122R21.051P-000".Pos_y07;
	::Camera:CameraPV.Output.Obj[7].Model AT %IB."VSC122R21.051P-000".Model08;
	::Camera:CameraPV.Output.Obj[7].Pos.X AT %ID."VSC122R21.051P-000".Pos_x08;
	::Camera:CameraPV.Output.Obj[7].Pos.Y AT %ID."VSC122R21.051P-000".Pos_y08;
END_VAR
```

### Config.mappmotioncfg - 5APC3100_KBU3_000/mappMotion/Config.mappmotioncfg
```
Element MappMotionConfiguration (Type=mappmotioncfg)
  Logger:
    SelectiveLogging = Used
      AdministrativeCommands = Suppressed
  Diagnostics:
    Snapshot = NotUsed
```

### Conveyer.axis - 5APC3100_KBU3_000/mappMotion/Conveyer/Conveyer.axis
```
Element conveyer1Ax (Type=axis)
  BaseType = LinearPeriodic
    MeasurementResolution = 0.001
    PeriodSettings:
      Period = 1870
  MovementLimits = InternalForPathControlledAxis
    Velocity:
      Velocity = 1000
    Acceleration:
      Acceleration = 1000
    Deceleration:
      Deceleration = 1000
    Jerk = Basic
Element conveyer2Ax (Type=axis)
  BaseType = LinearPeriodic
    MeasurementResolution = 0.001
    PeriodSettings:
      Period = 1870
  MovementLimits = InternalForPathControlledAxis
    Velocity:
      Velocity = 1000
    Acceleration:
      Acceleration = 1000
    Deceleration:
      Deceleration = 1000
    Jerk = Basic
Element repositoryAx (Type=axis)
  BaseType = LinearBounded
    MeasurementResolution = 0.001
  MovementLimits:
    Position:
      LowerLimit = -5
      UpperLimit = 505
    Velocity:
      Velocity = 600
    Acceleration:
      Acceleration = 2500
    Deceleration:
      Deceleration = 2500
```

### Conveyor.axisfeature - 5APC3100_KBU3_000/mappMotion/Conveyer/Conveyor.axisfeature
```
Element ProfGen (Type=axisfeature)
  Type = ProfGen
    JerkFilter = JerkLimited
```

### TrkPath.trackingpath - 5APC3100_KBU3_000/mappMotion/Conveyer/TrkPath.trackingpath
```
Element gTrackingPath_1 (Type=trackingpath)
  Type:
    MotionSource = Axis
      AxisRef = conveyer1Ax
    TrackingFrames:
      AutomaticCreation:
        Condition[1]:
          Distance = 350
          Activation = ProcessVariable
            ProcessVariableName = ::Mechanics:Cmd.Settings.Conveyor1.AutoFrameCreation.Enable
          Position:
            Translation:
              X = 175
              Z = 28
            Orientation:
              Angle3 = 180
          Attribute = 2#0001_0000
          UserData = CopyFromProcessVariable
            ProcessVariableName = ::Mechanics:UserDataEmptyPosForContainer
      AutomaticDeletion:
        Condition[1]:
          MinPosition = -50
          MaxPosition = 1870
        Condition[2] = AfterDesynchronization  // INSERTED FOR WORKING WITH VISION
          AxesGroupRef = gAxesGroup_D4r1100R_2
      UserData:
        Size = ProcessVariableReference
          ProcessVariableName = ::Mechanics:UserDataFullContainer
  SceneViewerObject:
    VisualRepresentation = Conveyor belt
      Dimensions:
        Length = 1870
        Width = 200
        Height = 50
      Translation:
        Y = -100
      Material = CyanMatte
Element gTrackingPath_2 (Type=trackingpath)
  Type:
    MaxPositionError = 3.0
    MotionSource = Axis
      AxisRef = conveyer2Ax
    TrackingFrames:
      AutomaticCreation:
        Condition[1]:
          Distance = 350
          Activation = ProcessVariable
            ProcessVariableName = ::Mechanics:Cmd.Settings.Conveyor2.AutoFrameCreation.Enable
          Position:
            Translation:
              Z = 27
          Attribute = 2#0000_0011
          UserData = CopyFromProcessVariable
            ProcessVariableName = ::Mechanics:UserDataEmptyContainer
      AutomaticDeletion:
        Condition[1]:
          MinPosition = -50
          MaxPosition = 1870
      UserData:
        Size = ProcessVariableReference
          ProcessVariableName = ::Mechanics:UserDataFullContainer
  SceneViewerObject:
    VisualRepresentation = Conveyor belt
      Dimensions:
        Length = 1870
        Width = 200
        Height = 50
      Translation:
        Y = -100
      Material = GreyMatte
Element gTrackingPath_3 (Type=trackingpath)
  Type:
    MotionSource:
      ProcessVariableName = ::Mechanics:Dummy_position
      NegativeOverflow = -10
      PositiveOverflow = 10
    TrackingFrames:
      UserData:
        Size = ProcessVariableReference
          ProcessVariableName = ::Mechanics:UserDataFullContainer
  SceneViewerObject:
    VisualRepresentation = Cuboid
      Dimensions:
        Length = 750
        Width = 200
        Height = 10
      Material = WhiteMatte
```

### AxGrp1.axesgroup - 5APC3100_KBU3_000/mappMotion/Delta1/AxGrp1.axesgroup
```
Element gAxesGroup_D4r1100R_1 (Type=axesgroup)
  Type = PathGenAxesGroup
    ProcessingTaskClass = 1
    PhysicalAxes:
      JointAxes:
        JointAxis[1]:
          AxisRef = delta1Q1
        JointAxis[2]:
          AxisRef = delta1Q2
        JointAxis[3]:
          AxisRef = delta1Q3
        JointAxis[4]:
          Name = QC
          AxisRef = delta1Qc
    MechanicalSystem:
      MechSysRef = delta1MechSys
    BasicSettings:
      GeometryPlanning:
        MaxCornerDeviation = 1
        MaxTangentialTransitionDeviation = 0.1
      TrajectoryPlanning:
        LimitCheckResolution:
          Time = 0.005
    AxesGroupFeatures:
      FeatureRef[1] = delta1Programs
      FeatureRef[2] = delta1Jogging
      FeatureRef[3] = delta1MFun
      FeatureRef[4] = delta1FrameHierarchy
      FeatureRef[5] = delta1Tracking
      FeatureRef[6] = delta1PathDef
      FeatureRef[7] = delta1Monitoring
      FeatureRef[8] = delta1WsMon
      FeatureRef[9] = delta1Tool
      FeatureRef[10] = Feature_TrkFrmSel_Delta_R1
```

### Axis1.axis - 5APC3100_KBU3_000/mappMotion/Delta1/Axis1.axis
```
Element delta1Q1 (Type=axis)
  BaseType = RotaryBounded
    MeasurementResolution = 0.001
    CountDirection = Inverse
  MovementLimits = InternalForPathControlledAxis
    Position:
      LowerLimit = -24
      UpperLimit = 85
    Velocity:
      Velocity = 2500
    Acceleration:
      Acceleration = 12000
    Deceleration:
      Deceleration = 12000
    Jerk = Basic
      Jerk = 120000
Element delta1Q2 (Type=axis)
  BaseType = RotaryBounded
    MeasurementResolution = 0.001
    CountDirection = Inverse
  MovementLimits = InternalForPathControlledAxis
    Position:
      LowerLimit = -24
      UpperLimit = 85
    Velocity:
      Velocity = 2500
    Acceleration:
      Acceleration = 12000
    Deceleration:
      Deceleration = 12000
    Jerk = Basic
      Jerk = 120000
Element delta1Q3 (Type=axis)
  BaseType = RotaryBounded
    MeasurementResolution = 0.001
    CountDirection = Inverse
  MovementLimits = InternalForPathControlledAxis
    Position:
      LowerLimit = -24
      UpperLimit = 85
    Velocity:
      Velocity = 2500
    Acceleration:
      Acceleration = 12000
    Deceleration:
      Deceleration = 12000
    Jerk = Basic
      Jerk = 120000
Element delta1Qc (Type=axis)
  BaseType = RotaryBounded
    MeasurementResolution = 0.001
    CountDirection = Inverse
  MovementLimits = InternalForPathControlledAxis
    Position:
      LowerLimit = -180
      UpperLimit = 180
    Velocity:
      Velocity = 720
    Acceleration:
      Acceleration = 7200
    Deceleration:
      Deceleration = 7200
    Jerk = Basic
      Jerk = 172000
```

### Feat1.axesgroupfeature - 5APC3100_KBU3_000/mappMotion/Delta1/Feat1.axesgroupfeature
```
Element delta1Programs (Type=axesgroupfeature)
  Type:
    DefaultLanguage = ST
    Location = User
      UserLocation[1]:
        FileDevice = RobotMotionPrgDir
Element delta1Jogging (Type=axesgroupfeature)
  Type = Jogging
Element delta1WsMon (Type=axesgroupfeature)
  Type = WorkspaceMonitoring
    WorkspaceRef = delta1Ws
Element delta1MFun (Type=axesgroupfeature)
  Type = MFunctions
Element delta1FrameHierarchy (Type=axesgroupfeature)
  Type = FrameHierarchy
Element delta1Tracking (Type=axesgroupfeature)
  Type = Tracking
    SynchronisationGeometry:
      CartesianRadius = 70
    MotionBehaviour:
      OutOfWorkspaceSynchronisation:
        Clearance = 25
Element delta1PathDef (Type=axesgroupfeature)
  Type = PathDefinitions
    PathDefinition[1]:
      Type:
        CalculatedIn = PCS
Element delta1Monitoring (Type=axesgroupfeature)
  Type = MonitoringElements
```

### Gripper1.tool - 5APC3100_KBU3_000/mappMotion/Delta1/Gripper1.tool
```
Element SingleGripper (Type=tool)
  ToolType = Robot
    Translation:
      X = 0
      Y = 0
      Z = -30
```

### MechSys1.mechanicalsystem - 5APC3100_KBU3_000/mappMotion/Delta1/MechSys1.mechanicalsystem
```
Element delta1MechSys (Type=mechanicalsystem)
  TypeIsReadOnly = 0
  Type = Delta
    SubtypeIsReadOnly = 0
    Subtype = 4AxesDeltaA
      SceneViewerObject = Generic
      DescriptionIsReadOnly = 0
      Description = Standard
        Dimensions:
          BasePlatform:
            CenterIsReadOnly = 0
            Center:
              X = 0.0
              Y = 0.0
              Z = -104
            ArmLinkPointIsReadOnly = 0
            Arm1LinkPoint:
              Angle = 0.0
              Radius = 100
              Z = 0
            Arm2LinkPoint:
              Angle = 120.0
              Radius = 100
              Z = 0
            Arm3LinkPoint:
              Angle = 240.0
              Radius = 100
              Z = 0
          Arms:
            ArmIsReadOnly = 0
            Arm1:
              UpperArmLength = 300
              LowerArmLength = 700
            Arm2:
              UpperArmLength = 300
              LowerArmLength = 700
            Arm3:
              UpperArmLength = 300
              LowerArmLength = 700
            LowerArmPairDistance = 0.0
          EndEffectorPlatform:
            ArmLinkPointIsReadOnly = 0
            Arm1LinkPoint:
              Radius = 50
              Z = 0.0
            Arm2LinkPoint:
              Radius = 50
              Z = 0.0
            Arm3LinkPoint:
              Radius = 50
              Z = 0.0
            TranslationToFlangeIsReadOnly = 0
            TranslationToFlange:
              X = 0.0
              Y = 0.0
              Z = -65
        Offsets:
          JointAxisIsReadOnly = 0
          JointAxis[1] = 0.0
          JointAxis[2] = 0.0
          JointAxis[3] = 0.0
          JointAxis[4] = 0.0
        CountDirections:
          JointAxisIsReadOnly = 0
          JointAxis[1] = Standard
          JointAxis[2] = Standard
          JointAxis[3] = Standard
          JointAxis[4] = Standard
      CoordinatesNames = Default
        XCoordinateName = X
        YCoordinateName = Y
        ZCoordinateName = Z
        CCoordinateName = C
      TcpOrientation:
        Frames = Used
      WireFrameModelIsReadOnly = 0
      WireFrameModel = Standard
        UpperArm1IsReadOnly = 0
        UpperArm1 = ConnectionLine
          DistanceMin = -1.79769313486231E308
          DistanceMax = 1.79769313486231E308
          Distance = 0.0
        LowerArm1IsReadOnly = 0
        LowerArm1 = ConnectionLine
          DistanceMin = -1.79769313486231E308
          DistanceMax = 1.79769313486231E308
          Distance = 0.0
        UpperArm2IsReadOnly = 0
        UpperArm2 = ConnectionLine
          DistanceMin = -1.79769313486231E308
          DistanceMax = 1.79769313486231E308
          Distance = 0.0
        LowerArm2IsReadOnly = 0
        LowerArm2 = ConnectionLine
          DistanceMin = -1.79769313486231E308
          DistanceMax = 1.79769313486231E308
          Distance = 0.0
        UpperArm3IsReadOnly = 0
        UpperArm3 = ConnectionLine
          DistanceMin = -1.79769313486231E308
          DistanceMax = 1.79769313486231E308
          Distance = 0.0
        LowerArm3IsReadOnly = 0
        LowerArm3 = ConnectionLine
          DistanceMin = -1.79769313486231E308
          DistanceMax = 1.79769313486231E308
          Distance = 0.0
        EndEffectorPlatformToFlangeIsReadOnly = 0
        EndEffectorPlatformToFlange = ConnectionLine
          DistanceMin = -1.79769313486231E308
          DistanceMax = 1.79769313486231E308
          Distance = 20
        FlangeToTcp = ConnectionLine
          DistanceMin = -1.79769313486231E308
          DistanceMax = 1.79769313486231E308
          Distance = 0.0
      DynamicModelIsReadOnly = 0
      DynamicModel = DynParTable
        TableRef
      InternalDynamicModelIsReadOnly = 0
      InternalDynamicModel = NotUsed
      DynamicLimits = DynParTables
        GearboxLimitsTableRef
        CrossSectionLimitsTableRef
      InternalDynamicLimits = NotUsed
      LoadDependentJerkLimitsIsReadOnly = 0
      LoadDependentJerkLimits = NotUsed
      CouplingsIsInvisible = 0
      JointAxesPositionLimits:
        JointAxisIsReadOnly = 0
        JointAxis[1] = UseAxisLimits
        JointAxis[2] = UseAxisLimits
        JointAxis[3] = UseAxisLimits
        JointAxis[4] = UseAxisLimits
      WorkingRangeIsReadOnly = 0
      WorkingRange = NotUsed
```

### TrkFrmSel1.axesgroupfeature - 5APC3100_KBU3_000/mappMotion/Delta1/TrkFrmSel1.axesgroupfeature
```
Element Feature_TrkFrmSel_Delta_R1 (Type=axesgroupfeature)
  Type = TrackingFrameSelection
    Selectors:
      Selector[1]:
        Name = Rob1_Pick_Conveyor1
        Strategy = MaximumXValueOnTrackingPath
        Filters:
          Filter[1]:
            TrackingPathRef[1] = gTrackingPath_1
          Filter[2] = SelectionArea
            Area[1]:
              Translation:
                X = -150
                Y = 100
                Z = -950
              Dimensions:
                Length = 350
                Width = 300
                Height = 300
        LockingAfterSelection = NoLocking
      Selector[2]:
        Name = Rob1_Place_Conveyor2
        Strategy = MaximumXValueOnTrackingPath
        Filters:
          Filter[1]:
            TrackingPathRef[1] = gTrackingPath_2  // ADD TRAKC VISION
          Filter[2] = SelectionArea
            Area[1]:
              Origin = MCS
              Translation:
                X = -450
                Y = -400
                Z = -950
              Dimensions:
                Length = 450
                Width = 300
                Height = 300
        LockingAfterSelection = NoLocking
      Selector[3]:
        Name = Rob1_PickPlace_Buffer
        Filters:
          Filter[1]:
            TrackingPathRef[1] = gTrackingPath_3
        LockingAfterSelection = NoLocking
```

### AxGrp2.axesgroup - 5APC3100_KBU3_000/mappMotion/Delta2/AxGrp2.axesgroup
```
Element gAxesGroup_D4r1100R_2 (Type=axesgroup)
  Type = PathGenAxesGroup
    ProcessingTaskClass = 1
    PhysicalAxes:
      JointAxes:
        JointAxis[1]:
          AxisRef = delta2Q1
        JointAxis[2]:
          AxisRef = delta2Q2
        JointAxis[3]:
          AxisRef = delta2Q3
        JointAxis[4]:
          Name = QC
          AxisRef = delta2Qc
    MechanicalSystem:
      MechSysRef = delta2MechSys
    BasicSettings:
      GeometryPlanning:
        MaxCornerDeviation = 1
        MaxTangentialTransitionDeviation = 0.1
      TrajectoryPlanning:
        LimitCheckResolution:
          Time = 0.005
    AxesGroupFeatures:
      FeatureRef[1] = delta2FrameHierarchy
      FeatureRef[2] = delta2Jogging
      FeatureRef[3] = delta2MFun
      FeatureRef[4] = delta2Programs
      FeatureRef[5] = delta2WsMon
      FeatureRef[6] = delta2Tool
      FeatureRef[7] = delta2Monitoring
      FeatureRef[8] = delta1Tracking
      FeatureRef[9] = delta1PathDef
      FeatureRef[10] = Feature_TrkFrmSel_Delta_R2
```

### Axis2.axis - 5APC3100_KBU3_000/mappMotion/Delta2/Axis2.axis
```
Element delta2Q1 (Type=axis)
  BaseType = RotaryBounded
    MeasurementResolution = 0.001
    CountDirection = Inverse
  MovementLimits = InternalForPathControlledAxis
    Position:
      LowerLimit = -24
      UpperLimit = 85
    Velocity:
      Velocity = 2500
    Acceleration:
      Acceleration = 12000
    Deceleration:
      Deceleration = 12000
    Jerk = Basic
      Jerk = 120000
Element delta2Q2 (Type=axis)
  BaseType = RotaryBounded
    MeasurementResolution = 0.001
    CountDirection = Inverse
  MovementLimits = InternalForPathControlledAxis
    Position:
      LowerLimit = -24
      UpperLimit = 85
    Velocity:
      Velocity = 2500
    Acceleration:
      Acceleration = 12000
    Deceleration:
      Deceleration = 12000
    Jerk = Basic
      Jerk = 120000
Element delta2Q3 (Type=axis)
  BaseType = RotaryBounded
    MeasurementResolution = 0.001
    CountDirection = Inverse
  MovementLimits = InternalForPathControlledAxis
    Position:
      LowerLimit = -24
      UpperLimit = 85
    Velocity:
      Velocity = 2500
    Acceleration:
      Acceleration = 12000
    Deceleration:
      Deceleration = 12000
    Jerk = Basic
      Jerk = 120000
Element delta2Qc (Type=axis)
  BaseType = RotaryBounded
    MeasurementResolution = 0.001
    CountDirection = Inverse
  MovementLimits = InternalForPathControlledAxis
    Position:
      LowerLimit = -180
      UpperLimit = 180
    Velocity:
      Velocity = 720
    Acceleration:
      Acceleration = 7200
    Deceleration:
      Deceleration = 7200
    Jerk = Basic
      Jerk = 172000
```

### Config_1.tool - 5APC3100_KBU3_000/mappMotion/Delta2/Config_1.tool
```
Element Tool_1 (Type=tool)
  ToolType:
    Translation:
      X = 25
      Y = 25
Element Tool_2 (Type=tool)
  ToolType:
    Translation:
      X = 25
      Y = -25
Element Tool_3 (Type=tool)
  ToolType:
    Translation:
      X = -25
      Y = -25
Element Tool_4 (Type=tool)
  ToolType:
    Translation:
      X = -25
      Y = 25
Element Tool_Cluster (Type=tool)
```

### Config_2.tooltable - 5APC3100_KBU3_000/mappMotion/Delta2/Config_2.tooltable
```
Element ToolTable_1 (Type=tooltable)
  Row[1]:
    ToolDataRef = Tool_1
  Row[2]:
    Index = 2
    ToolDataRef = Tool_2
  Row[3]:
    Index = 3
    ToolDataRef = Tool_3
  Row[4]:
    Index = 4
    ToolDataRef = Tool_4
  Row[5]:
    Index = 5
    ToolDataRef = Tool_Cluster
```

### Feat2.axesgroupfeature - 5APC3100_KBU3_000/mappMotion/Delta2/Feat2.axesgroupfeature
```
Element delta2Programs (Type=axesgroupfeature)
  Type:
    DefaultLanguage = ST
    Location = User
      UserLocation[1]:
        FileDevice = RobotMotionPrgDir
Element delta2Jogging (Type=axesgroupfeature)
  Type = Jogging
Element delta2WsMon (Type=axesgroupfeature)
  Type = WorkspaceMonitoring
    WorkspaceRef = delta2Ws
Element delta2MFun (Type=axesgroupfeature)
  Type = MFunctions
Element delta2FrameHierarchy (Type=axesgroupfeature)
  Type = FrameHierarchy
Element delta2Monitoring (Type=axesgroupfeature)
  Type = MonitoringElements
Element delta2Tool (Type=axesgroupfeature)
  Type = Tools
    Tools:
      ToolTable = ToolTable_1
      Index = 3
```

### Gripper2.tool - 5APC3100_KBU3_000/mappMotion/Delta2/Gripper2.tool
```
Element MultiGripper (Type=tool)
  ToolType = Robot
    Translation:
      X = -25
      Y = -25
      Z = -30
```

### MechSys2.mechanicalsystem - 5APC3100_KBU3_000/mappMotion/Delta2/MechSys2.mechanicalsystem
```
Element delta2MechSys (Type=mechanicalsystem)
  TypeIsReadOnly = 0
  Type = Delta
    SubtypeIsReadOnly = 0
    Subtype = 4AxesDeltaA
      SceneViewerObject = Generic
      DescriptionIsReadOnly = 0
      Description = Standard
        Dimensions:
          BasePlatform:
            CenterIsReadOnly = 0
            Center:
              X = 0.0
              Y = 0.0
              Z = -104
            ArmLinkPointIsReadOnly = 0
            Arm1LinkPoint:
              Angle = 180.0
              Radius = 100
              Z = 0.0
            Arm2LinkPoint:
              Angle = 300.0
              Radius = 100
              Z = 0.0
            Arm3LinkPoint:
              Angle = 420.0
              Radius = 100
              Z = 0.0
          Arms:
            ArmIsReadOnly = 0
            Arm1:
              UpperArmLength = 300
              LowerArmLength = 700
            Arm2:
              UpperArmLength = 300
              LowerArmLength = 700
            Arm3:
              UpperArmLength = 300
              LowerArmLength = 700
            LowerArmPairDistance = 0.0
          EndEffectorPlatform:
            ArmLinkPointIsReadOnly = 0
            Arm1LinkPoint:
              Radius = 50
              Z = 0.0
            Arm2LinkPoint:
              Radius = 50
              Z = 0.0
            Arm3LinkPoint:
              Radius = 50
              Z = 0.0
            TranslationToFlangeIsReadOnly = 0
            TranslationToFlange:
              X = 0.0
              Y = 0.0
              Z = -65
        Offsets:
          JointAxisIsReadOnly = 0
          JointAxis[1] = 0.0
          JointAxis[2] = 0.0
          JointAxis[3] = 0.0
          JointAxis[4] = 0.0
        CountDirections:
          JointAxisIsReadOnly = 0
          JointAxis[1] = Standard
          JointAxis[2] = Standard
          JointAxis[3] = Standard
          JointAxis[4] = Standard
      CoordinatesNames = Default
        XCoordinateName = X
        YCoordinateName = Y
        ZCoordinateName = Z
        CCoordinateName = C
      TcpOrientation:
        Frames = Used
      WireFrameModelIsReadOnly = 0
      WireFrameModel = Standard
        UpperArm1IsReadOnly = 0
        UpperArm1 = ConnectionLine
          DistanceMin = -1.79769313486231E308
          DistanceMax = 1.79769313486231E308
          Distance = 0.0
        LowerArm1IsReadOnly = 0
        LowerArm1 = ConnectionLine
          DistanceMin = -1.79769313486231E308
          DistanceMax = 1.79769313486231E308
          Distance = 0.0
        UpperArm2IsReadOnly = 0
        UpperArm2 = ConnectionLine
          DistanceMin = -1.79769313486231E308
          DistanceMax = 1.79769313486231E308
          Distance = 0.0
        LowerArm2IsReadOnly = 0
        LowerArm2 = ConnectionLine
          DistanceMin = -1.79769313486231E308
          DistanceMax = 1.79769313486231E308
          Distance = 0.0
        UpperArm3IsReadOnly = 0
        UpperArm3 = ConnectionLine
          DistanceMin = -1.79769313486231E308
          DistanceMax = 1.79769313486231E308
          Distance = 0.0
        LowerArm3IsReadOnly = 0
        LowerArm3 = ConnectionLine
          DistanceMin = -1.79769313486231E308
          DistanceMax = 1.79769313486231E308
          Distance = 0.0
        EndEffectorPlatformToFlangeIsReadOnly = 0
        EndEffectorPlatformToFlange = ConnectionLine
          DistanceMin = -1.79769313486231E308
          DistanceMax = 1.79769313486231E308
          Distance = 20
        FlangeToTcp = ConnectionLine
          DistanceMin = -1.79769313486231E308
          DistanceMax = 1.79769313486231E308
          Distance = 0.0
      DynamicModelIsReadOnly = 0
      DynamicModel = DynParTable
        TableRef
      InternalDynamicModelIsReadOnly = 0
      InternalDynamicModel = NotUsed
      DynamicLimits = DynParTables
        GearboxLimitsTableRef
        CrossSectionLimitsTableRef
      InternalDynamicLimits = NotUsed
      LoadDependentJerkLimitsIsReadOnly = 0
      LoadDependentJerkLimits = NotUsed
      CouplingsIsInvisible = 0
      JointAxesPositionLimits:
        JointAxisIsReadOnly = 0
        JointAxis[1] = UseAxisLimits
        JointAxis[2] = UseAxisLimits
        JointAxis[3] = UseAxisLimits
        JointAxis[4] = UseAxisLimits
      WorkingRangeIsReadOnly = 0
      WorkingRange = NotUsed
```

### TrkFrmSel2.axesgroupfeature - 5APC3100_KBU3_000/mappMotion/Delta2/TrkFrmSel2.axesgroupfeature
```
Element Feature_TrkFrmSel_Delta_R2 (Type=axesgroupfeature)
  Type = TrackingFrameSelection
    Selectors:
      Selector[1]:
        Name = Rob2_Pick_Conveyor2
        Strategy = MaximumXValueOnTrackingPath
        Filters:
          Filter[1]:
            TrackingPathRef[1] = gTrackingPath_2
          Filter[2] = SelectionArea
            Area[1]:
              Translation:
                X = -800
                Y = -400
                Z = -950
              Dimensions:
                Length = 800
                Width = 300
                Height = 300
        LockingAfterSelection = NoLocking
      Selector[2]:
        Name = Rob2_Place_Conveyor1
        Strategy = MinimumXValueOnTrackingPath
        Filters:
          Filter[1]:
            TrackingPathRef[1] = gTrackingPath_1
          Filter[2] = SelectionArea
            Area[1]:
              Origin = MCS
              Translation:
                X = -150
                Y = 100
                Z = -950
              Dimensions:
                Length = 700
                Width = 300
                Height = 300
        LockingAfterSelection = NoLocking
```

### Settings_1.vicfg - 5APC3100_KBU3_000/mappVision/Settings_1.vicfg
```
Element VisionSettings (Type=vicfg)
  ActivateVisualization = TRUE
  FileDeviceName
  Protocol = Unsecure
```

### viComp.visioncomponent - 5APC3100_KBU3_000/mappVision/viComp.visioncomponent
```
Element gCamera (Type=visioncomponent)
  VisionApplicationReference = ViApplication
  CompatibleVisionApplications:
    CompatibleVA[1] = ViApplication
```

## Logical view

Binary libraries used (declarations not repeated): Runtime, Operator, AsIecCon, astime, sys_lib, FileIO, AsMem, brsystem, AsBrStr, AsIOTime, standard, AsArSdm, AsBrWStr, AsHttp, AsZip, AsIO, AsIODiag, AsBrMath, MpBase, CoTrace 6.4.1, McBase 6.4.1, McAxGroup 6.6.1, McAcpAx 6.4.1, McAxis 6.4.1, McPathGen 6.6.1, McTrkPath 6.6.1, MpAxis 6.4.1, McProgInt 6.6.1, MpPick 6.7.2, McPureVAx 6.7.2, MpRobotics 6.6.1, MpTool 6.7.2, ViBase 6.0.0, AsARCfg, powerlnk, AsEPL, AsTCP, ArSsl, DataObj

### Globals.var
```iecst
VAR
	gVision : VisionCtrl_Type := (0);
	gMechanics : MechanicsCtrl_Type := (0);
END_VAR
VAR CONSTANT
	OBJECT_HEIGHT_mm : USINT := 27; (*mm*)
END_VAR
VAR
	SIMULATION_ACTIVE : BOOL := FALSE;
END_VAR
```

### Globals.typ
```iecst
(*Type for Mechanics ctrl structure*)

TYPE
	MechanicsStatus_Type : 	STRUCT
		Moving : BOOL;
		Homed : BOOL;
	END_STRUCT;
	MechanicsParam_Type : 	STRUCT
		CameraReady : BOOL;
	END_STRUCT;
	MechanicsCtrl_Type : 	STRUCT
		Status : MechanicsStatus_Type;
		Param : MechanicsParam_Type;
	END_STRUCT;
END_TYPE

(*Type for Vision ctrl structure*)

TYPE
	VisionCtrl_Type : 	STRUCT
		Param : VisionParam_Type;
		Status : VisionStatus_Type;
	END_STRUCT;
	VisionStatus_Type : 	STRUCT
		Configured : BOOL;
	END_STRUCT;
	VisionParam_Type : 	STRUCT
		MachineReadyAndHomed : BOOL;
	END_STRUCT;
END_TYPE
```


### Package Logical/Tasks - Including Source code and related objects

### Program Logical/Tasks/Mechanics (IEC) - Initialization,Homing and control of the conveyor and robots (PLC application task)

#### Main.st - Init, cyclic, exit code
```iecst
(**
 * Main Mechanics Control Program
 *
 * This program manages the complete pick-and-place system including:
 * - Two conveyor belts with automatic TrackingFrame creation
 * - Two robots (Robot 1: single object picker, Robot 2: container picker)
 * - System initialization, homing, and operational state management
 * - TrackingPath coordination and parameter management
 *
 * System Flow:
 * 0. Buffer: Provides initial objects for Robot 1 to pick from
 * 1. Conveyor 1: Feeds individual objects to Robot 1
 * 2. Robot 1: Picks objects and fills containers on Conveyor 2
 * 3. Robot 2: Transfers filled containers from Conveyor 2 back to Conveyor 1
 * 4. Buffer: Provides temporary storage when direct transfer isn't possible
 *
 * Purpose & Scope:
 * This demonstration program showcases how multiple mapp Robotics features can be integrated
 * to create a complete pick-and-place solution. The focus is on demonstrating feature integration
 * and process coordination rather than production-ready implementation.
 *
 * Note: This is a demonstration/training example and does not implement production-grade
 * safety protocols, error handling, or machine lifecycle management (power-up, homing,
 * shutdown procedures) that would be required for a real industrial application.
 *)

PROGRAM _INIT

	SIMULATION_ACTIVE := DiagCpuIsSimulated() OR DiagCpuIsARsim();

	// Initial process parameters
	Cmd.Settings.Conveyor1.AutoFrameCreation.Space := 200;
	Cmd.Settings.Conveyor2.AutoFrameCreation.Space := 200;
	Cmd.Settings.Conveyor1.Velocity := 60;
	Cmd.Settings.Conveyor2.Velocity := 60;

	// Robots
	MpRobotPar_1.ProgramName := 'PnpRobot1.st'; // Single object pick-and-place robot
	MpRobotPar_2.ProgramName := 'PnpRobot2.st'; // Container transfer robot

	Cmd.Settings.Robot1.AgilityReductionFactor := 1;
	Cmd.Settings.Robot1.SpeedLimitReductionFactor := 1;
	Cmd.Settings.Robot2.AgilityReductionFactor := 1;
	Cmd.Settings.Robot2.SpeedLimitReductionFactor := 1;

	MpRobot_1.MpLink := ADR(gAxesGroup_D4r1100R_1);
	MpRobot_1.Enable := TRUE;
	MpRobot_1.Parameters := ADR(MpRobotPar_1);
	MpRobot_1.Override := 100;

	MpRobot_2.MpLink := ADR(gAxesGroup_D4r1100R_2);
	MpRobot_2.Enable := TRUE;
	MpRobot_2.Parameters := ADR(MpRobotPar_2);
	MpRobot_2.Override := 100;

	// Conveyor belts
	MpAxisParConv1.Velocity := Cmd.Settings.Conveyor1.Velocity;
	MpAxisParConv2.Velocity := Cmd.Settings.Conveyor2.Velocity;
	MpAxisConv1.MpLink := ADR(conveyer1Ax);
	MpAxisConv1.Parameters := ADR(MpAxisParConv1);
	MpAxisConv1.Enable := TRUE;
	MpAxisConv2.MpLink := ADR(conveyer2Ax);
	MpAxisConv2.Parameters := ADR(MpAxisParConv2);
	MpAxisConv2.Enable := TRUE;
	StatusTrackingPath1.Enable := TRUE;
	StatusTrackingPath2.Enable := TRUE;
	StatusTrackingPath1.TrackingPath := ADR(gTrackingPath_1);
	StatusTrackingPath2.TrackingPath := ADR(gTrackingPath_2);

	// IMPORTANT: Coordinate system alignment between conveyors
	// TrackingPath_1 is 180° rotated relative to TrackingPath_2
	// To prevent robot rotation for each transfer from TrackingPath_1 to TrackingPath_2,
	// containers created on TrackingPath_1 are pre-rotated by 180°
	Cmd.Settings.Conveyor1.ContainerOrientation := 180; // Pre-rotation to match Path_2 orientation

	UseInternalPVs;

END_PROGRAM

(**
 * Main Cyclic Control Program
 *
 * Manages the complete system operation through a state machine:
 * 1. STARTUP - Wait for system readiness
 * 2. WAIT_FOR_POWER_AND_HOME - Wait for user command to start
 * 3. POWER - Power up all components
 * 4. HOME - Home all axes and robots
 * 5. READ_CURRENT_PARAMETERS - Initialize TrackingPath parameters
 * 6. RUN - Normal operation with continuous monitoring
 *)

PROGRAM _CYCLIC
	// Bridge for integrating the camera in the system
	CameraIntegration;

	// Synchronize user interface commands with robot/conveyor controls
	MotionProgramRob1.CleaningMachine := Cmd.CleanUpMode;

	IF gMechanics.Param.CameraReady THEN
		MpRobot_1.MoveProgram := Cmd.MoveProgramRobot1;
		MpRobot_2.MoveProgram := Cmd.MoveProgramRobot2;
		MpAxisConv1.MoveVelocity := Cmd.MoveConveyor1;
		MpAxisConv2.MoveVelocity := Cmd.MoveConveyor2;
	END_IF

	MpRobot_1.Stop := Cmd.Stop;
	MpRobot_2.Stop := Cmd.Stop;
	MpAxisConv1.Stop := Cmd.Stop;
	MpAxisConv2.Stop := Cmd.Stop;

	// Update robot performance parameters based on settings
	AgilityReductionInit;
	SpeedLimitReduction;

	CleaningProcess;

	(* Main state machine *)
	CASE Cmd.Info.State OF

		STARTUP:
			// Wait for all components to report ready status
			Cmd.Info.Status := 'Awaiting machine readiness before starting the system';
			IF MpAxisConv1.Info.ReadyToPowerOn AND MpAxisConv2.Info.ReadyToPowerOn AND MpRobot_1.Info.ReadyToPowerOn AND MpRobot_2.Info.ReadyToPowerOn  THEN
				Cmd.Info.State := WAIT_FOR_POWER_AND_HOME;
			END_IF

		WAIT_FOR_POWER_AND_HOME:
			// System ready - wait for operator command to begin startup sequence
			Cmd.Info.Status := 'Machine ready for power-up and homing!';
			IF Cmd.PowerAndHome THEN
				Cmd.Info.State := POWER;
			END_IF

		POWER:
			// Power up all components
			Cmd.Info.Status := 'Stuck here? Power-on failed, see log for details.';
			MpRobot_1.Power := TRUE;   // Power robot 1 drives
			MpRobot_2.Power := TRUE;   // Power robot 2 drives
			MpAxisConv1.Power := TRUE; // Power conveyor 1 drive
			MpAxisConv2.Power := TRUE; // Power conveyor 2 drive
			// Wait for all power-on confirmations before proceeding
			IF   MpAxisConv1.PowerOn AND MpAxisConv2.PowerOn AND MpRobot_1.PowerOn AND MpRobot_2.PowerOn THEN
				Cmd.Info.State := HOME;
			END_IF

		HOME:
			// Home all axes to establish reference positions
			IF SIMULATION_ACTIVE THEN
				// In simulation: Use direct homing (drives are simulated)
				SimHome;
			ELSE
				// Real hardware: Use absolute homing procedure
				MpRobot_1.Home := TRUE;
				MpRobot_2.Home := TRUE;

			END_IF
			MpAxisConv1.Home := TRUE;  // Home conveyor 1
			MpAxisConv2.Home := TRUE;  // Home conveyor 2

			// Wait for all homing operations to complete
			IF  MpAxisConv1.IsHomed AND MpAxisConv2.IsHomed AND MpRobot_1.IsHomed AND MpRobot_2.IsHomed THEN
				// Enable automatic tracking frame creation once homed
				Cmd.Settings.Conveyor1.AutoFrameCreation.Enable := TRUE;
				Cmd.Settings.Conveyor2.AutoFrameCreation.Enable := TRUE;
				Cmd.Info.State := READ_CURRENT_PARAMETERS;

				gMechanics.Status.Homed := TRUE;
			END_IF

		READ_CURRENT_PARAMETERS:

			// Read current automatic creation condition parameters configured for TrackingPath components

			IF StatusTrackingPath1.TrackingPathReady AND StatusTrackingPath2.TrackingPathReady THEN
				ReadgTrackingPath_1_param;
				ReadgTrackingPath_2_param;
			END_IF

			// Wait for parameter read operations to complete
			IF ProcessParam_AutCrtCond1TrkPath1.Done AND ProcessParam_AutCrtCond1TrkPath2.Done THEN
				// Reset function block execute flags
				ProcessParam_AutCrtCond1TrkPath1.Execute := FALSE;
				ProcessParam_AutCrtCond1TrkPath2.Execute := FALSE;

				// Update settings with values read from configuration
				Cmd.Settings.Conveyor1.AutoFrameCreation.Space := AutoCreateConditionParTrkPath1.Condition.DistanceBased.Distance;
				Cmd.Settings.Conveyor2.AutoFrameCreation.Space := AutoCreateConditionParTrkPath2.Condition.DistanceBased.Distance;

				Cmd.Info.Status := 'Machine Running';
				Cmd.Info.State := RUN;

			END_IF

		RUN:
			// Normal operation mode - continuous parameter monitoring and updates

			// Apply any changes to tracking path parameters during operation
			AdjustTrackingPath_1_distance;  // Update conveyor 1 frame spacing
			AdjustTrackingPath_2_distance;  // Update conveyor 2 frame spacing
			AdjustTrackingPath_1_Angle3;    // Update conveyor 1 container orientation

			// Dynamic conveyor velocity updates
			IF MpAxisParConv1.Velocity <> Cmd.Settings.Conveyor1.Velocity THEN
				MpAxisParConv1.Velocity := Cmd.Settings.Conveyor1.Velocity;
				MpAxisConv1.Update := TRUE;
				MpAxisConv1();
				MpAxisConv1.Update := FALSE;
			END_IF
			IF MpAxisParConv2.Velocity <> Cmd.Settings.Conveyor2.Velocity THEN
				MpAxisParConv2.Velocity := Cmd.Settings.Conveyor2.Velocity;
				MpAxisConv2.Update := TRUE;
				MpAxisConv2();
				MpAxisConv2.Update := FALSE;
			END_IF

			IF Cmd.Settings.Conveyor1.ContainerOrientation <= 0 OR Cmd.Settings.Conveyor1.ContainerOrientation >= 360 THEN
				Cmd.Info.Status := 'Please enter an orientation value greater than 0 and less than 360, robot 2 in error state';
				Cmd.Stop := TRUE;
			ELSE
				IF Cmd.Stop THEN
					Cmd.Stop := FALSE;
					// Note: MpRobot_.MoveProgram and MpAxisConv.MoveVelocity need manual restart after stop
				END_IF
			END_IF

	END_CASE

	MpRobot_1();
	MpRobot_2();

	MpAxisConv1();
	MpAxisConv2();

	ProcessParam_AutCrtCond1TrkPath1();
	ProcessParam_AutCrtCond1TrkPath2();

	StatusTrackingPath1();
	StatusTrackingPath2();

END_PROGRAM
```

#### GeneralActions.st
```iecst
ACTION UseInternalPVs :

	// Uses internal variables at least once to avoid unused variable warnings

	MotionProgramRob1;
	MotionProgramRob2;

	UserDataEmptyContainer;
	UserDataFullContainer;
	UserDataEmptyPosForContainer;

	repositoryAx;
	delta2Q1;
	delta2Q2;
	delta2Q3;
	delta2Qc;
	delta1Q1;
	delta1Q2;
	delta1Q3;
	delta1Qc;
	gPsm;
	Dummy_position;

END_ACTION

ACTION SimHome :

	MC_BR_GroupHome_0.AxesGroup := ADR(gAxesGroup_D4r1100R_1);
	MC_BR_GroupHome_1.AxesGroup := ADR(gAxesGroup_D4r1100R_2);
	MC_BR_GroupHome_0.Execute := TRUE;
	MC_BR_GroupHome_1.Execute := TRUE;
	FOR axIdx := 0 TO MAX_AXIS_IDX DO
		MC_BR_GroupHome_0.HomingMode[axIdx] := mcHOMING_DIRECT;
		MC_BR_GroupHome_0.Position[axIdx] := 0.0;
		MC_BR_GroupHome_1.HomingMode[axIdx] := mcHOMING_DIRECT;
		MC_BR_GroupHome_1.Position[axIdx] := 0.0;
	END_FOR;

	MC_BR_GroupHome_0();
	MC_BR_GroupHome_1();

END_ACTION

ACTION AgilityReductionInit:

	// During commissioning OR testing, it is advisable TO reduce the robot’s speed settings.
	// The provided code enables coordinated adjustment OF velocity, acceleration, AND jerk.
	// Remember TO declare any necessary variables, as they have been omitted in the example.

	MC_BR_GroupSetOverride_0_R1.Type := mcOVERRIDE_VELOCITY;
	MC_BR_GroupSetOverride_0_R1.Factor := Cmd.Settings.Robot1.AgilityReductionFactor;
	MC_BR_GroupSetOverride_0_R1.Enable := TRUE;

	MC_BR_GroupSetOverride_1_R1.Type := mcOVERRIDE_ACCELERATION;
	MC_BR_GroupSetOverride_1_R1.Factor := Cmd.Settings.Robot1.AgilityReductionFactor;
	MC_BR_GroupSetOverride_1_R1.Enable := TRUE;

	MC_BR_GroupSetOverride_2_R1.Type := mcOVERRIDE_JERK;
	MC_BR_GroupSetOverride_2_R1.Factor := Cmd.Settings.Robot1.AgilityReductionFactor;
	MC_BR_GroupSetOverride_2_R1.Enable := TRUE;

	MC_BR_GroupSetOverride_0_R1(AxesGroup := ADR(gAxesGroup_D4r1100R_1));
	MC_BR_GroupSetOverride_1_R1(AxesGroup := ADR(gAxesGroup_D4r1100R_1));
	MC_BR_GroupSetOverride_2_R1(AxesGroup := ADR(gAxesGroup_D4r1100R_1));

	MC_BR_GroupSetOverride_0_R2.Type := mcOVERRIDE_VELOCITY;
	MC_BR_GroupSetOverride_0_R2.Factor := Cmd.Settings.Robot2.AgilityReductionFactor;
	MC_BR_GroupSetOverride_0_R2.Enable := TRUE;

	MC_BR_GroupSetOverride_1_R2.Type := mcOVERRIDE_ACCELERATION;
	MC_BR_GroupSetOverride_1_R2.Factor := Cmd.Settings.Robot2.AgilityReductionFactor;
	MC_BR_GroupSetOverride_1_R2.Enable := TRUE;

	MC_BR_GroupSetOverride_2_R2.Type := mcOVERRIDE_JERK;
	MC_BR_GroupSetOverride_2_R2.Factor := Cmd.Settings.Robot2.AgilityReductionFactor;
	MC_BR_GroupSetOverride_2_R2.Enable := TRUE;

	MC_BR_GroupSetOverride_0_R2(AxesGroup := ADR(gAxesGroup_D4r1100R_2));
	MC_BR_GroupSetOverride_1_R2(AxesGroup := ADR(gAxesGroup_D4r1100R_2));
	MC_BR_GroupSetOverride_2_R2(AxesGroup := ADR(gAxesGroup_D4r1100R_2));

END_ACTION

ACTION SpeedLimitReduction:

	MC_BR_GroupSetOverride_0_R1.Type := mcOVERRIDE_VELOCITY;
	MC_BR_GroupSetOverride_0_R1.Factor := Cmd.Settings.Robot1.SpeedLimitReductionFactor;
	MC_BR_GroupSetOverride_0_R1.Enable := TRUE;
	MC_BR_GroupSetOverride_0_R1(AxesGroup := ADR(gAxesGroup_D4r1100R_1));

	MC_BR_GroupSetOverride_0_R2.Type := mcOVERRIDE_VELOCITY;
	MC_BR_GroupSetOverride_0_R2.Factor := Cmd.Settings.Robot2.SpeedLimitReductionFactor;
	MC_BR_GroupSetOverride_0_R2.Enable := TRUE;
	MC_BR_GroupSetOverride_0_R2(AxesGroup := ADR(gAxesGroup_D4r1100R_2));

END_ACTION

ACTION CameraIntegration :
	 // When mechanics is homed, allow vision to start/configure
	IF gMechanics.Status.Homed THEN
		gVision.Param.MachineReadyAndHomed := TRUE;
	END_IF
	// When vision is configured, notify mechanics that the camera is ready
	IF gVision.Status.Configured THEN
		gMechanics.Param.CameraReady := TRUE;
	END_IF
END_ACTION
```

#### TrkPathParActions.st
```iecst
// Reads the current auto-create condition parameters for Tracking Path 1 from the configuration.
ACTION ReadgTrackingPath_1_param:

	ProcessParam_AutCrtCond1TrkPath1.Execute := TRUE;
	ProcessParam_AutCrtCond1TrkPath1.Component := ADR(gTrackingPath_1);
	ProcessParam_AutCrtCond1TrkPath1.AdvancedParameters.Name := 'Condition 1';
	ProcessParam_AutCrtCond1TrkPath1.DataAddress := ADR(AutoCreateConditionParTrkPath1);
	ProcessParam_AutCrtCond1TrkPath1.DataType := mcCFG_TRK_PATH_AUT_CRT_COND;
	ProcessParam_AutCrtCond1TrkPath1.Mode := mcPPM_READ;

END_ACTION

// Reads the current auto-create condition parameters for Tracking Path 2 from the configuration.
ACTION ReadgTrackingPath_2_param:

	ProcessParam_AutCrtCond1TrkPath2.Execute := TRUE;
	ProcessParam_AutCrtCond1TrkPath2.Component := ADR(gTrackingPath_2);
	ProcessParam_AutCrtCond1TrkPath2.AdvancedParameters.Name := 'Condition 1';
	ProcessParam_AutCrtCond1TrkPath2.DataAddress := ADR(AutoCreateConditionParTrkPath2);
	ProcessParam_AutCrtCond1TrkPath2.DataType := mcCFG_TRK_PATH_AUT_CRT_COND;
	ProcessParam_AutCrtCond1TrkPath2.Mode := mcPPM_READ;

END_ACTION

// Checks if the distance parameter for Tracking Path 1 needs updating.
// If so, updates the value and writes it back to the controller.
ACTION AdjustTrackingPath_1_distance:

	IF AutoCreateConditionParTrkPath1.Condition.DistanceBased.Distance <> Cmd.Settings.Conveyor1.AutoFrameCreation.Space THEN
		AutoCreateConditionParTrkPath1.Condition.DistanceBased.Distance := Cmd.Settings.Conveyor1.AutoFrameCreation.Space;
		ProcessParam_AutCrtCond1TrkPath1.Execute := TRUE;
		ProcessParam_AutCrtCond1TrkPath1.Component := ADR(gTrackingPath_1);
		ProcessParam_AutCrtCond1TrkPath1.AdvancedParameters.Name := 'Condition 1';
		ProcessParam_AutCrtCond1TrkPath1.DataAddress := ADR(AutoCreateConditionParTrkPath1);
		ProcessParam_AutCrtCond1TrkPath1.DataType := mcCFG_TRK_PATH_AUT_CRT_COND;
		ProcessParam_AutCrtCond1TrkPath1.Mode := mcPPM_WRITE;
		ProcessParam_AutCrtCond1TrkPath1();
		ProcessParam_AutCrtCond1TrkPath1.Execute := FALSE;
	END_IF

END_ACTION

// Checks if the distance parameter for Tracking Path 2 needs updating.
// If so, updates the value and writes it back to the controller.
ACTION AdjustTrackingPath_2_distance:

	IF AutoCreateConditionParTrkPath2.Condition.DistanceBased.Distance <> Cmd.Settings.Conveyor2.AutoFrameCreation.Space THEN
		AutoCreateConditionParTrkPath2.Condition.DistanceBased.Distance := Cmd.Settings.Conveyor2.AutoFrameCreation.Space;
		ProcessParam_AutCrtCond1TrkPath2.Execute := TRUE;
		ProcessParam_AutCrtCond1TrkPath2.Component := ADR(gTrackingPath_2);
		ProcessParam_AutCrtCond1TrkPath2.AdvancedParameters.Name := 'Condition 1';
		ProcessParam_AutCrtCond1TrkPath2.DataAddress := ADR(AutoCreateConditionParTrkPath2);
		ProcessParam_AutCrtCond1TrkPath2.DataType := mcCFG_TRK_PATH_AUT_CRT_COND;
		ProcessParam_AutCrtCond1TrkPath2.Mode := mcPPM_WRITE;
		ProcessParam_AutCrtCond1TrkPath2();
		ProcessParam_AutCrtCond1TrkPath2.Execute := FALSE;
	END_IF

END_ACTION

// Writes the updated frame position parameters for Tracking Path 1 to the controller.
ACTION UpdateTrackingPath_1_FramePos:

	ProcessParam_AutCrtCond1TrkPath1.Execute := TRUE;
	ProcessParam_AutCrtCond1TrkPath1.Component := ADR(gTrackingPath_1);
	ProcessParam_AutCrtCond1TrkPath1.AdvancedParameters.Name := 'Condition 1';
	ProcessParam_AutCrtCond1TrkPath1.DataAddress := ADR(AutoCreateConditionParTrkPath1);
	ProcessParam_AutCrtCond1TrkPath1.DataType := mcCFG_TRK_PATH_AUT_CRT_COND;
	ProcessParam_AutCrtCond1TrkPath1.Mode := mcPPM_WRITE;
	ProcessParam_AutCrtCond1TrkPath1();
	ProcessParam_AutCrtCond1TrkPath1.Execute := FALSE;

END_ACTION

// Checks if the orientation angle (Angle3) for Tracking Path 1 needs updating.
// If so, updates the value and writes the new frame position to the controller.
ACTION AdjustTrackingPath_1_Angle3:

	IF AutoCreateConditionParTrkPath1.Condition.DistanceBased.Position.Orientation.Angle3 <> Cmd.Settings.Conveyor1.ContainerOrientation THEN
		AutoCreateConditionParTrkPath1.Condition.DistanceBased.Position.Orientation.Angle3 := Cmd.Settings.Conveyor1.ContainerOrientation ;
		UpdateTrackingPath_1_FramePos;
	END_IF

END_ACTION

// During cleaning, only automatic frame creation for conveyor 2 is disabled.
// This ensures objects are placed at origin after cleaning.
// Stopping frame creation on conveyor 1 would require checking that all objects are back,
// which is application-specific and not implemented here.

ACTION CleaningProcess:
	// Ensure the system is in RUN state to avoid interfering with automatic frame creation,
	// which must wait until the conveyor homing process is completed.
	IF Cmd.Info.State = RUN THEN

		// If the cleaning machine is active, disable automatic frame creation of tracking path 2
		IF Cmd.CleanUpMode THEN
			Cmd.Settings.Conveyor2.AutoFrameCreation.Enable := FALSE;
			// Otherwise, if automatic frame creation is currently disabled, enable it
		ELSIF Cmd.Settings.Conveyor2.AutoFrameCreation.Enable = FALSE THEN
			Cmd.Settings.Conveyor2.AutoFrameCreation.Enable := TRUE;
		END_IF

	END_IF
END_ACTION
```

#### Types.typ - Local data types
```iecst
TYPE
	CommandType : 	STRUCT
		PowerAndHome : BOOL;
		MoveConveyor1 : BOOL;
		MoveConveyor2 : BOOL;
		MoveProgramRobot1 : BOOL;
		MoveProgramRobot2 : BOOL;
		Settings : CmdSettingsType;
		Info : InfoType;
		Stop : BOOL;
		CleanUpMode : BOOL; (*once TRUE the robots will start to put the object back to the container*)
	END_STRUCT;
	RobotSettingsType : 	STRUCT
		AgilityReductionFactor : REAL; (*Reduces the velocity, acceleration and jerk limits (path limit and axes limit). Value range 0 to 1. This value must not be changed during program run.*)
		SpeedLimitReductionFactor : REAL; (*Reduces the velocity limit (path limit and axes limit). Value range 0 to 1. This value can also be changed during program run.*)
	END_STRUCT;
	TrackingFrameCreationType : 	STRUCT
		Enable : BOOL;
		Space : LREAL;
	END_STRUCT;
	Conveyor1SettingsType : 	STRUCT
		Velocity : REAL;
		AutoFrameCreation : TrackingFrameCreationType;
		ContainerOrientation : REAL; (*The orientation of Container 1 is defined relative to the coordinate system of Tracking Path 1. A value of 180° indicates a 180-degree rotation around the Z-axis from the original orientation of Tracking Path 1.

The robot allows rotation values strictly between 0° and 360°—that is, values must be greater than 0° and less than 360°. Both 0° and 360° are not included in the allowed range to avoid ambiguity*)
	END_STRUCT;
	Conveyor2SettingsType : 	STRUCT
		Velocity : REAL;
		AutoFrameCreation : TrackingFrameCreationType;
	END_STRUCT;
	CmdSettingsType : 	STRUCT
		Conveyor1 : Conveyor1SettingsType;
		Conveyor2 : Conveyor2SettingsType;
		Robot1 : RobotSettingsType;
		Robot2 : RobotSettingsType;
	END_STRUCT;
	StateType :
		(
		STARTUP,
		WAIT_FOR_POWER_AND_HOME,
		POWER,
		HOME,
		READ_CURRENT_PARAMETERS,
		RUN
		);
	InfoType : 	STRUCT
		Status : STRING[120];
		State : StateType;
	END_STRUCT;
END_TYPE
```

#### Variables.var - Local variables
```iecst
(*Command interface*)
VAR
	Cmd : CommandType;
END_VAR
(*Robot and conveyor FBs*)
VAR
	MpRobot_1 : MpDelta4Axis;
	MpRobot_2 : MpDelta4Axis;
	MpRobotPar_1 : MpDelta4AxisParType;
	MpRobotPar_2 : MpDelta4AxisParType;
	MpAxisConv1 : MpAxisBasic;
	MpAxisConv2 : MpAxisBasic;
	MpAxisParConv1 : MpAxisBasicParType;
	MpAxisParConv2 : MpAxisBasicParType;
END_VAR
(*Update automatic TrackingFrame creation *)
VAR
	ProcessParam_AutCrtCond1TrkPath1 : MC_BR_ProcessParam;
	ProcessParam_AutCrtCond1TrkPath2 : MC_BR_ProcessParam;
	AutoCreateConditionParTrkPath1 : McCfgTrkPathAutCrtCondType;
	AutoCreateConditionParTrkPath2 : McCfgTrkPathAutCrtCondType;
END_VAR
(*Insert your comment here.*)
VAR
	StatusTrackingPath1 : MC_BR_TrackingPathReadStatus;
	StatusTrackingPath2 : MC_BR_TrackingPathReadStatus;
END_VAR
(*Motion Program data structures*)
VAR
	MotionProgramRob1 : RobotMotionProgramType := (0);
	MotionProgramRob2 : RobotMotionProgramType := (0);
END_VAR
(*Initialized variables for TrackingFrame user data*)
VAR
	UserDataEmptyContainer : {REDUND_UNREPLICABLE} TrackingFrameUserDataType := (SubFramesVisu:=[2((Pos:=(X:=0,Y:=0))),(Pos:=(X:=0,Y:=50)),(Pos:=(X:=50,Y:=0)),(Pos:=(X:=50,Y:=50))],PositionType:=ContainerPosition,ContainerPositionData:=(PositionFilled:=TRUE,ContainedPositions:=[(PositionFilled:=FALSE,ObjectType:=Red,SyncPosUp:=(Pos:=(X:=0,Y:=0,Z:=10+OBJECT_HEIGHT_mm)),SyncPosDown:=(Pos:=(X:=0,Y:=0,Z:=0))),(PositionFilled:=FALSE,ObjectType:=Red,SyncPosUp:=(Pos:=(X:=0,Y:=50,Z:=10+OBJECT_HEIGHT_mm)),SyncPosDown:=(Pos:=(X:=0,Y:=50,Z:=0))),(PositionFilled:=FALSE,ObjectType:=Black,SyncPosUp:=(Pos:=(X:=50,Y:=0,Z:=10+OBJECT_HEIGHT_mm)),SyncPosDown:=(Pos:=(X:=50,Y:=0,Z:=0))),(PositionFilled:=FALSE,ObjectType:=Black,SyncPosUp:=(Pos:=(X:=50,Y:=50,Z:=10+OBJECT_HEIGHT_mm)),SyncPosDown:=(Pos:=(X:=50,Y:=50,Z:=0)))],SyncPosUp:=(Pos:=(Z:=10+OBJECT_HEIGHT_mm))));
	UserDataFullContainer : {REDUND_UNREPLICABLE} TrackingFrameUserDataType := (SubFramesVisu:=[(Pos:=(X:=0,Y:=0)),(Pos:=(X:=0,Y:=0),Attribute:=RedObjectPhysicallyPresent),(Pos:=(X:=0,Y:=50),Attribute:=RedObjectPhysicallyPresent),(Pos:=(X:=50,Y:=0),Attribute:=BlackObjectPhysicallyPresent),(Pos:=(X:=50,Y:=50),Attribute:=BlackObjectPhysicallyPresent)],PositionType:=ContainerPosition,ContainerPositionData:=(PositionFilled:=TRUE,ContainedPositions:=[(PositionFilled:=TRUE,ObjectType:=Red,SyncPosUp:=(Pos:=(X:=0,Y:=0,Z:=10+OBJECT_HEIGHT_mm)),SyncPosDown:=(Pos:=(X:=0,Y:=0,Z:=0))),(PositionFilled:=TRUE,ObjectType:=Red,SyncPosUp:=(Pos:=(X:=0,Y:=50,Z:=10+OBJECT_HEIGHT_mm)),SyncPosDown:=(Pos:=(X:=0,Y:=50,Z:=0))),(PositionFilled:=TRUE,ObjectType:=Black,SyncPosUp:=(Pos:=(X:=50,Y:=0,Z:=10+OBJECT_HEIGHT_mm)),SyncPosDown:=(Pos:=(X:=50,Y:=0,Z:=0))),(PositionFilled:=TRUE,ObjectType:=Black,SyncPosUp:=(Pos:=(X:=50,Y:=50,Z:=10+OBJECT_HEIGHT_mm)),SyncPosDown:=(Pos:=(X:=50,Y:=50,Z:=0)))],SyncPosUp:=(Pos:=(Z:=10+OBJECT_HEIGHT_mm))));
	UserDataEmptyPosForContainer : {REDUND_UNREPLICABLE} TrackingFrameUserDataType := (SubFramesVisu:=[2((Pos:=(X:=0,Y:=0))),(Pos:=(X:=0,Y:=50)),(Pos:=(X:=50,Y:=0)),(Pos:=(X:=50,Y:=50))],PositionType:=ContainerPosition,ContainerPositionData:=(PositionFilled:=FALSE,ContainedPositions:=[(PositionFilled:=FALSE,ObjectType:=Red,SyncPosUp:=(Pos:=(X:=0,Y:=0,Z:=10+OBJECT_HEIGHT_mm)),SyncPosDown:=(Pos:=(X:=0,Y:=0,Z:=0))),(PositionFilled:=FALSE,ObjectType:=Red,SyncPosUp:=(Pos:=(X:=0,Y:=50,Z:=10+OBJECT_HEIGHT_mm)),SyncPosDown:=(Pos:=(X:=0,Y:=50,Z:=0))),(PositionFilled:=FALSE,ObjectType:=Black,SyncPosUp:=(Pos:=(X:=50,Y:=0,Z:=10+OBJECT_HEIGHT_mm)),SyncPosDown:=(Pos:=(X:=50,Y:=0,Z:=0))),(PositionFilled:=FALSE,ObjectType:=Black,SyncPosUp:=(Pos:=(X:=50,Y:=50,Z:=10+OBJECT_HEIGHT_mm)),SyncPosDown:=(Pos:=(X:=50,Y:=50,Z:=0)))],SyncPosUp:=(Pos:=(Z:=10+OBJECT_HEIGHT_mm))));
END_VAR
(*Variable for tracking pah link*)
VAR
	Dummy_position : LREAL := 0.0;
END_VAR
(*Direct homing for simulation mode*)
VAR
	MC_BR_GroupHome_0 : MC_BR_GroupHome_15;
	MC_BR_GroupHome_1 : MC_BR_GroupHome_15;
	axIdx : USINT;
END_VAR
VAR CONSTANT
	MAX_AXIS_IDX : USINT := 4;
END_VAR
(*Changing robot override*)
VAR
	MC_BR_GroupSetOverride_0_R1 : MC_BR_GroupSetOverride := (0);
	MC_BR_GroupSetOverride_1_R1 : MC_BR_GroupSetOverride := (0);
	MC_BR_GroupSetOverride_2_R1 : MC_BR_GroupSetOverride := (0);
	MC_BR_GroupSetOverride_0_R2 : MC_BR_GroupSetOverride := (0);
	MC_BR_GroupSetOverride_1_R2 : MC_BR_GroupSetOverride := (0);
	MC_BR_GroupSetOverride_2_R2 : MC_BR_GroupSetOverride := (0);
END_VAR
```

### Program Logical/Tasks/Camera (IEC) - Manages creating new TrackingFrames based on camera detections: filters results, converts pixel to millimeter coordinates, and submits valid frames to the TrackingPath.

#### Main.st - Init, cyclic, exit code
```iecst
(**
 * Vision Manager Main Program
 * This program manages the complete vision pipeline for a pick-and-place system, including:
 * - Axis-based image acquisition synchronized to conveyor motion
 * - Camera configuration and readiness checks
 * - Detection filtering (Derive position and color of the physical objects from the detected shapes)
 * - Pixel-to-millimeter coordinate transformation
 * - TrackingFrame creation and submission to the TrackingPath
 *
 * System Flow:

 * 0. WAITING_FOR_SYSTEM_READY: Verify camera/module OK and machine homed; initialize camera; enable acquisition
 * 1. NEXT_CAPTURE_PENDING: Detect a new completed acquisition; request current frames for de-duplication checks
 * 2. WAITING_VF: Wait for the vision function to finish image processing
 * 3. DETECTED_OBJECT_FRAME_CREATION: Filter detections, transform to mm, reject near-existing frames, stage frames, submit batch
 * 4. RESETTING_FB: Reset function blocks and buffers; return to NEXT_CAPTURE_PENDING
 *
 * Purpose & Scope:
 * This demonstration module shows how to integrate camera acquisition, detection filtering,
 * and tracking frame creation into a conveyor-based workflow, ensuring only valid,
 * de-duplicated detections are promoted TO TrackingFrames.
 *
 * Note: This is a demonstration/training example and does not implement production-grade
 * safety protocols, error handling, or machine lifecycle management (power-up, homing,
 * shutdown procedures) that would be required for a real industrial application.
 *)

PROGRAM _INIT

	MC_ReadActualPosition_Mot1(Axis := ADR(conveyer1Ax), Enable := TRUE);
	MC_BR_DetectedObjFramesCreat.TrackingPath := ADR(gTrackingPath_1);

	GetFramesInfoInitialization;

	ViBaseAxisBasedAcquisition_Fb.Enable := FALSE;
	ViBaseAxisBasedAcquisition_Fb.MpLink := ADR(gCamera);
	ViBaseAxisBasedAcquisition_Fb.AcquisitionParameters.Period := 70; // it will take a picture every 80mm

	gVision.Param.MachineReadyAndHomed := FALSE;

END_PROGRAM

PROGRAM _CYCLIC

	ViBaseAxisBasedAcquisition_Fb();
	MC_BR_DetectedObjFramesCreat();
	TrackingPathGetFramesPos_Fb();

	CASE VisionState OF

		WAITING_FOR_SYSTEM_READY:
			IF CameraPV.Status.CameraStatus = 0 AND CameraPV.Status.ModuleOk AND gVision.Param.MachineReadyAndHomed THEN
				ViBaseAxisBasedAcquisition_Fb.Enable := TRUE; // enable the acquisition, when the axis is home and ready
				CameraInitialization;
				gVision.Status.Configured := TRUE;
				VisionState := NEXT_CAPTURE_PENDING;
			END_IF;

		NEXT_CAPTURE_PENDING:
			IF LastAcquisitionCount <> CameraPV.Status.CompletedAcquisitionCount   THEN
				MC_ReadActualPosition_Mot1();
				TrackingPathGetFramesPos_Fb.Execute := TRUE;
				VisionState := WAITING_VF;
			END_IF

		WAITING_VF:
			IF NOT CameraPV.Status.ImageProcessingActive THEN
				VisionState := DETECTED_OBJECT_FRAME_CREATION;
			END_IF

		DETECTED_OBJECT_FRAME_CREATION:

			IF TrackingPathGetFramesPos_Fb.Done AND NOT CameraPV.Status.ImageProcessingActive THEN
				IF  CameraPV.Output.NumObjFound > 0  THEN
					TrackingPathGetFramesPos_Fb.Execute := FALSE;
					LastAcquisitionCount := CameraPV.Status.CompletedAcquisitionCount;
					NumbersNewFrame := 0;
					CameraOutputFiltering;

					FOR i := 0 TO (CameraOutputFiltered.NumObjFound-1)   DO

						// Affine transformation with translation term (pixel -> mm)
						// Matrix components:
						// X_mm = (X_pixel * a11) + (Y_pixel * a12) + X_Translation_mm
						// Y_mm = (X_pixel * a21) + (Y_pixel * a22) + Y_Translation_mm
						//
						// From  matrix:
						// a11 = -0.17952376
						// a12 = -0.0015347
						// a21 =  0.00212256
						// a22 =  0.18369122
						// X_Translation_mm = 1102.51630312;
						// Y_Translation_mm = -89.82579615;

						CreateNewFrame := TRUE;

						Pos_mm[i].X :=((DINT_TO_LREAL(CameraOutputFiltered.Obj[i].Pos.X) * (-0.17952376))
						+ (DINT_TO_LREAL(CameraOutputFiltered.Obj[i].Pos.Y) * 0.00212256 ))/100 + 1102.51630312;

						Pos_mm[i].Y := ((DINT_TO_LREAL(CameraOutputFiltered.Obj[i].Pos.X) * (-0.0015347))
						+ (DINT_TO_LREAL(CameraOutputFiltered.Obj[i].Pos.Y) * 0.18369122))/100  -89.82579615;

						// This loop prevents creating duplicate frames. It calculates the Euclidean distance between the newly detected object and all existing ones.
						// IF any existing frame is closer than OBJECT_MIN_DIST, the new detection is rejected setting CreateNewFrame to FALSE
						FOR j := 0 TO TrackingPathGetFramesPos_Fb.TrackingFrameCount DO

							Distance := SQRT(
							brmpow(LREAL_TO_REAL(FramesInfo[j].CurrentPosition.X - Pos_mm[i].X), 2) +
							brmpow(LREAL_TO_REAL(FramesInfo[j].CurrentPosition.Y - Pos_mm[i].Y), 2)
							);
							IF Distance < OBJECT_MIN_DIST THEN
								CreateNewFrame := FALSE;
								EXIT;
							END_IF
						END_FOR

						// assign all the necessary Position information to the array McTrkFramesDetectedObjArray
						IF CreateNewFrame THEN
							McTrkFramesDetectedObjArray[NumbersNewFrame].Translation.X := Pos_mm[i].X;
							McTrkFramesDetectedObjArray[NumbersNewFrame].Translation.Y := Pos_mm[i].Y;
							McTrkFramesDetectedObjArray[NumbersNewFrame].Translation.Z := OBJECT_HEIGHT_mm;
							McTrkFramesDetectedObjArray[NumbersNewFrame].Orientation.Angle3 := 180;

							IF CameraOutputFiltered.Obj[i].Model = 2 THEN
								McTrkFramesDetectedObjArray[NumbersNewFrame].Attribute := HasBlackObj;
								McTrkFramesDetectedObjArray[NumbersNewFrame].UserDataAddress := ADR(UserDataSingleItemObjectBlack);
							ELSE
								McTrkFramesDetectedObjArray[NumbersNewFrame].Attribute := HasRedObj;
								McTrkFramesDetectedObjArray[NumbersNewFrame].UserDataAddress := ADR(UserDataSingleItemObjectRed);
							END_IF

							McTrkFramesDetectedObjArray[NumbersNewFrame].LatchedPath.Position := MC_ReadActualPosition_Mot1.Position;
							NumbersNewFrame := NumbersNewFrame + 1;
						END_IF

					END_FOR;

					IF NumbersNewFrame > 0 THEN
						MC_BR_DetectedObjFramesCreat.Parameters.DataAddress := ADR(McTrkFramesDetectedObjArray);
						MC_BR_DetectedObjFramesCreat.Parameters.NumberOfFrames := NumbersNewFrame;
						MC_BR_DetectedObjFramesCreat.Execute := TRUE;
					END_IF

					VisionState := RESETTING_VARIABLES;

				ELSE
					LastAcquisitionCount := CameraPV.Status.CompletedAcquisitionCount;
					TrackingPathGetFramesPos_Fb.Execute := FALSE;
					VisionState := NEXT_CAPTURE_PENDING;
				END_IF
			END_IF

		RESETTING_VARIABLES:

			IF MC_BR_DetectedObjFramesCreat.Done OR  NumbersNewFrame = 0 THEN
				TrackingPathGetFramesPos_Fb.Execute := FALSE;
				brsmemset(ADR(McTrkFramesDetectedObjArray),0,SIZEOF(McTrkFramesDetectedObjArray));
				MC_BR_DetectedObjFramesCreat.Execute := FALSE;
				brsmemset(ADR(CameraOutputFiltered),0,SIZEOF(CameraOutputFiltered));
				VisionState := NEXT_CAPTURE_PENDING;
			END_IF

	END_CASE

END_PROGRAM

PROGRAM _EXIT

	(* Cleanup and resource deallocation *)

	MC_ReadActualPosition_Mot1.Enable := FALSE;
	MC_ReadActualPosition_Mot1(); // Recall the FB

	ViBaseAxisBasedAcquisition_Fb.Enable := FALSE;
	ViBaseAxisBasedAcquisition_Fb();

END_PROGRAM
```

#### Types.typ - Local data types
```iecst
TYPE
	CameraParam_Type : 	STRUCT
		GainLevel : USINT;
		SetFocus : UINT;
		FlashSegment : USINT;
		FlashColor : USINT;
		ExposureTime : UDINT;
	END_STRUCT;
	CameraStatus_Type : 	STRUCT
		ModuleOk : BOOL;
		CameraStatus : UDINT;
		CompletedAcquisitionCount : USINT;
		ImageProcessingActive : BOOL;
	END_STRUCT;
	Camera_Type : 	STRUCT
		Status : CameraStatus_Type;
		Param : CameraParam_Type;
		Output : VF_Output_Type;
		Input : VF_Input_Type;
	END_STRUCT;
	CoordinatePixel_Type : 	STRUCT
		X : DINT;
		Y : DINT;
	END_STRUCT;
	Coordinate_mm_Type : 	STRUCT
		X : LREAL;
		Y : LREAL;
	END_STRUCT;
	ObjInfo_Type : 	STRUCT  (*information regarding the object found*)
		Pos : CoordinatePixel_Type;
		Orient : REAL;
		Model : USINT;
	END_STRUCT;
	VF_Input_Type : 	STRUCT
		EnableVF : BOOL; (*Input for enabling the VisionFunction*)
		NumSearchMax : USINT;
	END_STRUCT;
	VF_Output_Type : 	STRUCT
		NumObjFound : USINT;
		Obj : ARRAY[0..MaxObjectDetectable]OF ObjInfo_Type;
	END_STRUCT;
	VisionState_Enum :
		(
		WAITING_FOR_SYSTEM_READY, (*in this state camera triggering is waiting the correct configuration of the axis connected*)
		NEXT_CAPTURE_PENDING,
		WAITING_VF,
		DETECTED_OBJECT_FRAME_CREATION, (*Retrieves existing frames on the conveyor, filters raw camera detections (via CameraOutputFiltering),
converts kept detections from pixels to millimeters with an affine transform, and creates new tracking frames only
if each candidate is at least OBJECT_MIN_DIST away from all already-present frames.
Assigns attributes/user data BY color (BLACK/RED) and latches the current conveyor position before submitting the batch TO the tracking path.*)
		RESETTING_VARIABLES
		);
END_TYPE
```
